C03658=1180.309,271.886,-67.108,-177.055,7.451,148.555
C03659=1180.314,271.637,-67.079,-177.057,7.448,148.555
C03660=1180.318,271.389,-67.051,-177.060,7.446,148.555
C03661=1180.323,271.140,-67.023,-177.063,7.443,148.555
C03662=1180.327,270.893,-66.995,-177.066,7.440,148.555
C03663=1180.331,270.644,-66.967,-177.068,7.438,148.555
C03664=1180.336,270.396,-66.938,-177.071,7.435,148.555
C03665=1180.340,270.147,-66.910,-177.073,7.432,148.555
C03666=1180.345,269.899,-66.882,-177.076,7.430,148.556
C03667=1180.348,269.651,-66.854,-177.078,7.427,148.556
C03668=1180.354,269.402,-66.825,-177.081,7.424,148.556
C03669=1180.357,269.154,-66.797,-177.083,7.421,148.556
C03670=1180.362,268.906,-66.769,-177.086,7.418,148.556
C03671=1180.366,268.657,-66.741,-177.089,7.416,148.556
C03672=1180.371,268.408,-66.714,-177.092,7.413,148.556
C03673=1180.375,268.160,-66.685,-177.094,7.411,148.556
C03674=1180.380,267.912,-66.657,-177.097,7.408,148.556
C03675=1180.383,267.663,-66.629,-177.099,7.405,148.556
C03676=1180.388,267.415,-66.601,-177.102,7.403,148.556
C03677=1180.393,267.167,-66.573,-177.104,7.400,148.556
C03678=1180.397,266.919,-66.545,-177.107,7.397,148.556
C03679=1180.401,266.670,-66.518,-177.109,7.394,148.557
C03680=1180.406,266.421,-66.489,-177.112,7.392,148.557
C03681=1180.410,266.173,-66.461,-177.115,7.389,148.557
C03682=1180.414,265.925,-66.433,-177.117,7.387,148.557
C03683=1180.419,265.676,-66.406,-177.120,7.384,148.557
C03684=1180.424,265.428,-66.378,-177.123,7.381,148.557
C03685=1180.427,265.179,-66.349,-177.125,7.379,148.557
C03686=1180.432,264.932,-66.322,-177.128,7.376,148.557
C03687=1180.436,264.682,-66.294,-177.131,7.373,148.557
C03688=1180.441,264.434,-66.266,-177.133,7.371,148.558
C03689=1180.445,264.186,-66.238,-177.136,7.368,148.558
C03690=1180.449,263.937,-66.211,-177.139,7.365,148.558
C03691=1180.454,263.689,-66.183,-177.141,7.363,148.558
C03692=1180.459,263.441,-66.154,-177.144,7.360,148.558
C03693=1180.463,263.192,-66.127,-177.146,7.357,148.558
C03694=1180.467,262.944,-66.099,-177.149,7.355,148.558
C03695=1180.472,262.671,-66.069,-177.152,7.352,148.558
C03696=1180.477,262.398,-66.038,-177.154,7.349,148.558
C03697=1180.481,262.125,-66.008,-177.157,7.346,148.558
C03698=1180.486,261.852,-65.978,-177.160,7.343,148.559
C03699=1180.490,261.604,-65.950,-177.163,7.340,148.559
C03700=1180.495,261.355,-65.922,-177.166,7.337,148.559
C03701=1180.500,261.107,-65.894,-177.168,7.335,148.559
C03702=1180.504,260.858,-65.867,-177.171,7.332,148.559
C03703=1180.508,260.610,-65.839,-177.173,7.330,148.559
C03704=1180.513,260.362,-65.812,-177.176,7.327,148.559
C03705=1180.517,260.113,-65.784,-177.179,7.324,148.559
C03706=1180.521,259.864,-65.757,-177.181,7.322,148.559
C03707=1180.526,259.617,-65.729,-177.184,7.319,148.559
C03708=1180.530,259.367,-65.702,-177.187,7.317,148.560
C03709=1180.534,259.119,-65.675,-177.189,7.314,148.560
C03710=1180.539,258.871,-65.647,-177.192,7.311,148.560
C03711=1180.543,258.623,-65.620,-177.194,7.309,148.560
C03712=1180.547,258.374,-65.592,-177.197,7.306,148.560
C03713=1180.552,258.125,-65.564,-177.200,7.304,148.560
C03714=1180.556,257.877,-65.537,-177.202,7.302,148.560
C03715=1180.561,257.629,-65.510,-177.205,7.299,148.560
C03716=1180.565,257.380,-65.482,-177.208,7.296,148.560
C03717=1180.569,257.131,-65.455,-177.210,7.293,148.560
C03718=1180.574,256.884,-65.427,-177.213,7.291,148.561
C03719=1180.578,256.635,-65.400,-177.215,7.289,148.561
C03720=1180.582,256.386,-65.373,-177.218,7.286,148.561
C03721=1180.587,256.138,-65.345,-177.221,7.283,148.561
C03722=1180.591,255.889,-65.318,-177.223,7.281,148.561
C03723=1180.596,255.641,-65.291,-177.226,7.278,148.561
C03724=1180.600,255.392,-65.264,-177.228,7.276,148.561
C03725=1180.604,255.144,-65.236,-177.231,7.273,148.561
C03726=1180.609,254.895,-65.209,-177.234,7.270,148.562
C03727=1180.614,254.647,-65.182,-177.236,7.268,148.562
C03728=1180.618,254.398,-65.155,-177.239,7.265,148.562
C03729=1180.623,254.150,-65.128,-177.241,7.263,148.562
C03730=1180.626,253.902,-65.100,-177.244,7.260,148.562
C03731=1180.631,253.653,-65.073,-177.247,7.257,148.562
C03732=1180.635,253.405,-65.046,-177.249,7.255,148.562
C03733=1180.640,253.156,-65.019,-177.252,7.252,148.562
C03734=1180.645,252.908,-64.992,-177.255,7.250,148.563
C03735=1180.649,252.658,-64.964,-177.257,7.247,148.563
C03736=1180.653,252.410,-64.937,-177.260,7.245,148.563
C03737=1180.657,252.162,-64.911,-177.262,7.242,148.563
C03738=1180.662,251.913,-64.884,-177.265,7.240,148.563
C03739=1180.667,251.665,-64.857,-177.268,7.237,148.563
C03740=1180.671,251.417,-64.829,-177.270,7.234,148.563
C03741=1180.676,251.168,-64.802,-177.273,7.233,148.564
C03742=1180.680,250.920,-64.775,-177.276,7.230,148.564
C03743=1180.684,250.671,-64.748,-177.278,7.227,148.564
C03744=1180.688,250.423,-64.721,-177.281,7.224,148.564
C03745=1180.693,250.174,-64.694,-177.284,7.222,148.564
C03746=1180.697,249.926,-64.667,-177.286,7.220,148.564
C03747=1180.702,249.677,-64.641,-177.289,7.217,148.564
C03748=1180.707,249.428,-64.614,-177.291,7.215,148.565
C03749=1180.711,249.180,-64.587,-177.294,7.212,148.565
C03750=1180.715,248.932,-64.560,-177.296,7.210,148.565
C03751=1180.720,248.683,-64.533,-177.299,7.207,148.565
C03752=1180.724,248.435,-64.506,-177.302,7.205,148.565
C03753=1180.728,248.186,-64.480,-177.304,7.202,148.565
C03754=1180.732,247.937,-64.452,-177.307,7.199,148.565
C03755=1180.737,247.689,-64.425,-177.310,7.197,148.566
C03756=1180.741,247.441,-64.399,-177.313,7.194,148.566
C03757=1180.746,247.191,-64.373,-177.315,7.192,148.566
C03758=1180.751,246.943,-64.345,-177.318,7.189,148.566
C03759=1180.755,246.695,-64.319,-177.320,7.187,148.566
C03760=1180.759,246.446,-64.292,-177.323,7.184,148.566
C03761=1180.764,246.198,-64.265,-177.326,7.182,148.567
C03762=1180.768,245.949,-64.239,-177.328,7.180,148.567
C03763=1180.773,245.700,-64.212,-177.330,7.177,148.567
C03764=1180.777,245.452,-64.185,-177.334,7.175,148.567
C03765=1180.781,245.204,-64.159,-177.336,7.173,148.567
C03766=1180.786,244.955,-64.132,-177.339,7.170,148.567
C03767=1180.790,244.706,-64.106,-177.342,7.167,148.567
C03768=1180.795,244.458,-64.079,-177.344,7.165,148.568
C03769=1180.799,244.209,-64.053,-177.347,7.162,148.568
C03770=1180.804,243.961,-64.026,-177.349,7.160,148.568
C03771=1180.808,243.712,-63.999,-177.352,7.157,148.568
C03772=1180.813,243.463,-63.973,-177.355,7.155,148.568
C03773=1180.817,243.215,-63.946,-177.357,7.152,148.568
C03774=1180.821,242.967,-63.920,-177.360,7.150,148.568
C03775=1180.826,242.718,-63.893,-177.363,7.147,148.569
C03776=1180.830,242.469,-63.867,-177.365,7.145,148.569
C03777=1180.835,242.220,-63.840,-177.368,7.142,148.569
C03778=1180.840,241.973,-63.814,-177.370,7.141,148.569
C03779=1180.844,241.724,-63.787,-177.373,7.138,148.569
C03780=1180.848,241.475,-63.761,-177.376,7.136,148.570
C03781=1180.852,241.227,-63.735,-177.379,7.133,148.570
C03782=1180.857,240.978,-63.709,-177.381,7.131,148.570
C03783=1180.861,240.730,-63.682,-177.384,7.128,148.570
C03784=1180.866,240.481,-63.656,-177.386,7.126,148.570
C03785=1180.870,240.233,-63.629,-177.389,7.123,148.570
C03786=1180.875,239.984,-63.603,-177.392,7.121,148.571
C03787=1180.879,239.735,-63.577,-177.394,7.118,148.571
C03788=1180.884,239.486,-63.550,-177.397,7.116,148.571
C03789=1180.889,239.238,-63.525,-177.400,7.113,148.571
C03790=1180.893,238.990,-63.498,-177.402,7.111,148.571
C03791=1180.898,238.741,-63.472,-177.405,7.109,148.571
C03792=1180.902,238.493,-63.446,-177.407,7.106,148.572
C03793=1180.906,238.244,-63.420,-177.410,7.104,148.572
C03794=1180.911,237.995,-63.393,-177.413,7.102,148.572
C03795=1180.915,237.747,-63.367,-177.415,7.100,148.572
C03796=1180.920,237.497,-63.341,-177.418,7.097,148.572
C03797=1180.924,237.249,-63.315,-177.421,7.095,148.573
C03798=1180.928,237.001,-63.289,-177.423,7.092,148.573
C03799=1180.933,236.729,-63.261,-177.427,7.089,148.573
C03800=1180.938,236.458,-63.231,-177.429,7.087,148.573
C03801=1180.943,236.186,-63.203,-177.432,7.085,148.573
C03802=1180.948,235.915,-63.175,-177.435,7.082,148.573
C03803=1180.953,235.666,-63.149,-177.437,7.080,148.574
C03804=1180.957,235.417,-63.123,-177.440,7.077,148.574
C03805=1180.961,235.168,-63.097,-177.443,7.075,148.574
C03806=1180.965,234.920,-63.071,-177.446,7.072,148.574
C03807=1180.970,234.671,-63.044,-177.448,7.070,148.575
C03808=1180.975,234.423,-63.019,-177.451,7.067,148.575
C03809=1180.979,234.174,-62.993,-177.454,7.065,148.575
C03810=1180.983,233.925,-62.967,-177.456,7.062,148.575
C03811=1180.988,233.677,-62.940,-177.458,7.060,148.575
C03812=1180.993,233.429,-62.915,-177.462,7.058,148.575
C03813=1180.997,233.180,-62.889,-177.464,7.056,148.576
C03814=1181.001,232.931,-62.863,-177.467,7.054,148.576
C03815=1181.006,232.682,-62.838,-177.469,7.051,148.576
C03816=1181.011,232.434,-62.812,-177.472,7.049,148.576
C03817=1181.015,232.185,-62.786,-177.475,7.046,148.576
C03818=1181.020,231.936,-62.760,-177.477,7.044,148.577
C03819=1181.024,231.688,-62.734,-177.480,7.041,148.577
C03820=1181.028,231.440,-62.708,-177.483,7.039,148.577
C03821=1181.033,231.191,-62.683,-177.485,7.037,148.577
C03822=1181.038,230.942,-62.656,-177.488,7.035,148.577
C03823=1181.042,230.693,-62.631,-177.490,7.032,148.578
C03824=1181.047,230.445,-62.605,-177.493,7.030,148.578
C03825=1181.051,230.196,-62.579,-177.496,7.028,148.578
C03826=1181.055,229.948,-62.554,-177.499,7.025,148.578
C03827=1181.060,229.700,-62.528,-177.501,7.023,148.578
C03828=1181.064,229.451,-62.503,-177.504,7.021,148.579
C03829=1181.068,229.202,-62.477,-177.506,7.018,148.579
C03830=1181.073,228.953,-62.452,-177.509,7.016,148.579
C03831=1181.078,228.704,-62.426,-177.512,7.013,148.579
C03832=1181.082,228.456,-62.401,-177.515,7.012,148.580
C03833=1181.087,228.208,-62.375,-177.517,7.009,148.580
C03834=1181.092,227.958,-62.349,-177.520,7.007,148.580
C03835=1181.096,227.710,-62.323,-177.522,7.005,148.580
C03836=1181.101,227.462,-62.298,-177.525,7.002,148.580
C03837=1181.105,227.213,-62.272,-177.528,7.000,148.581
C03838=1181.109,226.964,-62.246,-177.530,6.998,148.581
C03839=1181.114,226.715,-62.222,-177.533,6.995,148.581
C03840=1181.119,226.466,-62.196,-177.536,6.993,148.581
C03841=1181.123,226.218,-62.170,-177.539,6.991,148.581
C03842=1181.128,225.969,-62.145,-177.541,6.989,148.582
C03843=1181.131,225.721,-62.120,-177.544,6.987,148.582
C03844=1181.136,225.472,-62.095,-177.546,6.984,148.582
C03845=1181.140,225.223,-62.069,-177.549,6.982,148.582
C03846=1181.145,224.975,-62.043,-177.552,6.979,148.582
C03847=1181.149,224.727,-62.018,-177.554,6.977,148.583
C03848=1181.154,224.477,-61.993,-177.557,6.975,148.583
C03849=1181.159,224.229,-61.968,-177.560,6.972,148.583
C03850=1181.163,223.980,-61.942,-177.562,6.971,148.583
C03851=1181.168,223.731,-61.917,-177.565,6.968,148.584
C03852=1181.172,223.483,-61.891,-177.568,6.966,148.584
C03853=1181.177,223.234,-61.866,-177.570,6.964,148.584
C03854=1181.182,222.985,-61.841,-177.573,6.961,148.584
C03855=1181.185,222.737,-61.816,-177.576,6.959,148.585
C03856=1181.190,222.489,-61.790,-177.578,6.957,148.585
C03857=1181.195,222.239,-61.765,-177.581,6.954,148.585
C03858=1181.199,221.990,-61.740,-177.583,6.952,148.585
C03859=1181.204,221.742,-61.715,-177.586,6.951,148.585
C03860=1181.208,221.493,-61.689,-177.589,6.948,148.586
C03861=1181.213,221.244,-61.665,-177.592,6.946,148.586
C03862=1181.217,220.996,-61.639,-177.594,6.944,148.586
C03863=1181.222,220.747,-61.614,-177.597,6.941,148.586
C03864=1181.226,220.498,-61.589,-177.600,6.939,148.587
C03865=1181.231,220.250,-61.564,-177.602,6.936,148.587
C03866=1181.235,220.001,-61.539,-177.605,6.934,148.587
C03867=1181.240,219.753,-61.514,-177.608,6.933,148.587
C03868=1181.244,219.503,-61.489,-177.610,6.930,148.587
C03869=1181.249,219.255,-61.463,-177.613,6.928,148.588
C03870=1181.254,219.006,-61.438,-177.616,6.926,148.588
C03871=1181.258,218.757,-61.414,-177.618,6.923,148.588
C03872=1181.262,218.509,-61.388,-177.621,6.921,148.589
C03873=1181.267,218.260,-61.364,-177.623,6.919,148.589
C03874=1181.271,218.011,-61.339,-177.627,6.917,148.589
C03875=1181.276,217.763,-61.314,-177.629,6.915,148.589
C03876=1181.280,217.514,-61.288,-177.631,6.913,148.589
C03877=1181.285,217.265,-61.264,-177.635,6.910,148.590
C03878=1181.290,217.017,-61.239,-177.637,6.908,148.590
C03879=1181.294,216.768,-61.214,-177.639,6.906,148.590
C03880=1181.299,216.519,-61.189,-177.643,6.903,148.590
C03881=1181.303,216.270,-61.165,-177.645,6.901,148.591
C03882=1181.308,216.022,-61.139,-177.648,6.899,148.591
C03883=1181.312,215.773,-61.114,-177.651,6.897,148.591
C03884=1181.317,215.524,-61.090,-177.653,6.895,148.591
C03885=1181.322,215.275,-61.065,-177.656,6.893,148.592
C03886=1181.325,215.027,-61.040,-177.659,6.890,148.592
C03887=1181.330,214.778,-61.016,-177.661,6.888,148.592
C03888=1181.335,214.529,-60.991,-177.664,6.886,148.592
C03889=1181.339,214.280,-60.967,-177.667,6.884,148.593
C03890=1181.344,214.032,-60.941,-177.669,6.882,148.593
C03891=1181.348,213.783,-60.917,-177.672,6.880,148.593
C03892=1181.353,213.534,-60.892,-177.674,6.878,148.594
C03893=1181.357,213.285,-60.867,-177.677,6.875,148.594
C03894=1181.362,213.037,-60.843,-177.680,6.873,148.594
C03895=1181.367,212.788,-60.818,-177.682,6.871,148.594
C03896=1181.371,212.539,-60.793,-177.685,6.868,148.594
C03897=1181.376,212.291,-60.768,-177.688,6.867,148.595
C03898=1181.380,212.042,-60.744,-177.691,6.865,148.595
C03899=1181.385,211.793,-60.719,-177.693,6.862,148.595
C03900=1181.389,211.544,-60.695,-177.696,6.860,148.596
C03901=1181.394,211.296,-60.671,-177.699,6.858,148.596
C03902=1181.398,211.047,-60.646,-177.701,6.856,148.596
C03903=1181.403,210.776,-60.619,-177.704,6.854,148.596
C03904=1181.408,210.506,-60.593,-177.707,6.851,148.597
C03905=1181.413,210.235,-60.566,-177.710,6.849,148.597
C03906=1181.418,209.965,-60.539,-177.713,6.846,148.597
C03907=1181.422,209.717,-60.515,-177.715,6.844,148.597
C03908=1181.427,209.467,-60.490,-177.718,6.843,148.598
C03909=1181.431,209.219,-60.466,-177.721,6.840,148.598
C03910=1181.436,208.970,-60.441,-177.723,6.838,148.598
C03911=1181.441,208.722,-60.417,-177.726,6.836,148.598
C03912=1181.445,208.472,-60.392,-177.729,6.834,148.599
C03913=1181.450,208.224,-60.368,-177.731,6.831,148.599
C03914=1181.454,207.975,-60.345,-177.734,6.829,148.599
C03915=1181.459,207.726,-60.320,-177.737,6.828,148.600
C03916=1181.463,207.477,-60.295,-177.739,6.826,148.600
C03917=1181.468,207.228,-60.271,-177.742,6.823,148.600
C03918=1181.473,206.980,-60.247,-177.745,6.821,148.600
C03919=1181.477,206.732,-60.223,-177.748,6.819,148.601
C03920=1181.482,206.482,-60.198,-177.750,6.816,148.601
C03921=1181.486,206.234,-60.173,-177.753,6.815,148.601
C03922=1181.491,205.985,-60.150,-177.756,6.813,148.601
C03923=1181.496,205.736,-60.125,-177.758,6.811,148.602
C03924=1181.500,205.487,-60.101,-177.761,6.808,148.602
C03925=1181.504,205.238,-60.077,-177.764,6.806,148.602
C03926=1181.509,204.990,-60.052,-177.766,6.804,148.603
C03927=1181.514,204.741,-60.029,-177.769,6.802,148.603
C03928=1181.518,204.492,-60.005,-177.772,6.800,148.603
C03929=1181.523,204.243,-59.980,-177.774,6.798,148.603
C03930=1181.527,203.994,-59.956,-177.777,6.796,148.604
C03931=1181.532,203.745,-59.932,-177.779,6.794,148.604
C03932=1181.536,203.497,-59.908,-177.782,6.791,148.604
C03933=1181.542,203.248,-59.884,-177.785,6.789,148.605
C03934=1181.545,202.999,-59.859,-177.788,6.788,148.605
C03935=1181.550,202.750,-59.836,-177.790,6.786,148.605
C03936=1181.554,202.502,-59.812,-177.793,6.784,148.605
C03937=1181.560,202.253,-59.787,-177.796,6.781,148.606
C03938=1181.564,202.004,-59.764,-177.798,6.779,148.606
C03939=1181.569,201.755,-59.740,-177.801,6.777,148.606
C03940=1181.573,201.507,-59.716,-177.803,6.775,148.606
C03941=1181.577,201.257,-59.692,-177.807,6.773,148.607
C03942=1181.582,201.009,-59.667,-177.809,6.771,148.607
C03943=1181.587,200.760,-59.644,-177.812,6.769,148.607
C03944=1181.591,200.511,-59.620,-177.814,6.767,148.608
C03945=1181.596,200.263,-59.596,-177.817,6.765,148.608
C03946=1181.600,200.014,-59.572,-177.820,6.763,148.608
C03947=1181.605,199.765,-59.548,-177.822,6.761,148.608
C03948=1181.610,199.516,-59.525,-177.825,6.759,148.609
C03949=1181.614,199.267,-59.500,-177.828,6.757,148.609
C03950=1181.619,199.018,-59.476,-177.831,6.754,148.609
C03951=1181.623,198.769,-59.452,-177.833,6.752,148.610
C03952=1181.628,198.520,-59.429,-177.836,6.750,148.610
C03953=1181.632,198.272,-59.405,-177.838,6.749,148.610
C03954=1181.637,198.023,-59.382,-177.841,6.747,148.611
C03955=1181.641,197.775,-59.358,-177.844,6.744,148.611
C03956=1181.646,197.525,-59.334,-177.846,6.742,148.611
C03957=1181.651,197.276,-59.311,-177.849,6.740,148.611
C03958=1181.655,197.028,-59.287,-177.852,6.739,148.612
C03959=1181.660,196.779,-59.263,-177.854,6.737,148.612
C03960=1181.665,196.530,-59.239,-177.857,6.735,148.612
C03961=1181.670,196.281,-59.215,-177.860,6.732,148.613
C03962=1181.674,196.032,-59.192,-177.863,6.730,148.613
C03963=1181.679,195.784,-59.168,-177.865,6.728,148.613
C03964=1181.683,195.535,-59.145,-177.868,6.727,148.614
C03965=1181.688,195.286,-59.121,-177.870,6.724,148.614
C03966=1181.692,195.037,-59.097,-177.873,6.722,148.614
C03967=1181.697,194.788,-59.073,-177.876,6.720,148.614
C03968=1181.701,194.539,-59.050,-177.879,6.718,148.615
C03969=1181.706,194.290,-59.026,-177.881,6.716,148.615
C03970=1181.710,194.041,-59.003,-177.883,6.714,148.615
C03971=1181.715,193.792,-58.979,-177.886,6.713,148.616
C03972=1181.719,193.545,-58.956,-177.889,6.710,148.616
C03973=1181.724,193.296,-58.933,-177.892,6.708,148.616
C03974=1181.729,193.047,-58.909,-177.895,6.706,148.617
C03975=1181.734,192.798,-58.886,-177.897,6.704,148.617
C03976=1181.738,192.549,-58.863,-177.900,6.702,148.617
C03977=1181.743,192.300,-58.839,-177.902,6.701,148.617
C03978=1181.747,192.051,-58.815,-177.905,6.698,148.618
C03979=1181.752,191.802,-58.792,-177.908,6.696,148.618
C03980=1181.757,191.553,-58.769,-177.911,6.694,148.618
C03981=1181.761,191.304,-58.745,-177.913,6.692,148.619
C03982=1181.766,191.055,-58.722,-177.916,6.691,148.619
C03983=1181.771,190.807,-58.698,-177.918,6.689,148.619
C03984=1181.774,190.558,-58.675,-177.922,6.686,148.620
C03985=1181.779,190.309,-58.652,-177.924,6.684,148.620
C03986=1181.784,190.060,-58.628,-177.927,6.683,148.620
C03987=1181.789,189.811,-58.605,-177.929,6.680,148.620
C03988=1181.793,189.562,-58.582,-177.932,6.679,148.621
C03989=1181.798,189.313,-58.558,-177.934,6.677,148.621
C03990=1181.803,189.065,-58.536,-177.937,6.675,148.622
C03991=1181.807,188.816,-58.512,-177.940,6.672,148.622
C03992=1181.812,188.567,-58.489,-177.943,6.671,148.622
C03993=1181.817,188.318,-58.466,-177.945,6.669,148.622
C03994=1181.821,188.069,-58.442,-177.948,6.667,148.623
C03995=1181.825,187.820,-58.420,-177.951,6.665,148.623
C03996=1181.830,187.571,-58.396,-177.953,6.663,148.623
C03997=1181.835,187.322,-58.373,-177.956,6.661,148.624
C03998=1181.840,187.073,-58.350,-177.959,6.660,148.624
C03999=1181.844,186.825,-58.327,-177.962,6.657,148.624
C04000=1181.849,186.576,-58.304,-177.964,6.655,148.625
C04001=1181.853,186.327,-58.280,-177.967,6.653,148.625
C04002=1181.858,186.078,-58.257,-177.969,6.651,148.625
C04003=1181.862,185.829,-58.234,-177.972,6.650,148.626
C04004=1181.867,185.580,-58.211,-177.975,6.648,148.626
C04005=1181.872,185.332,-58.188,-177.977,6.646,148.626
C04006=1181.876,185.082,-58.166,-177.980,6.644,148.627
C04007=1181.881,184.813,-58.140,-177.983,6.642,148.627
C04008=1181.887,184.543,-58.115,-177.986,6.640,148.627
C04009=1181.891,184.274,-58.091,-177.989,6.638,148.628
C04010=1181.897,184.004,-58.066,-177.992,6.635,148.628
C04011=1181.901,183.755,-58.042,-177.995,6.634,148.628
C04012=1181.905,183.506,-58.020,-177.997,6.632,148.629
C04013=1181.910,183.257,-57.997,-177.999,6.630,148.629
C04014=1181.915,183.008,-57.974,-178.002,6.628,148.629
C04015=1181.919,182.760,-57.951,-178.005,6.626,148.630
C04016=1181.924,182.511,-57.928,-178.007,6.624,148.630
C04017=1181.928,182.261,-57.906,-178.010,6.623,148.630
C04018=1181.933,182.012,-57.882,-178.013,6.620,148.631
C04019=1181.938,181.764,-57.859,-178.016,6.618,148.631
C04020=1181.943,181.515,-57.837,-178.019,6.616,148.631
C04021=1181.947,181.265,-57.814,-178.021,6.615,148.632
C04022=1181.951,181.017,-57.791,-178.024,6.613,148.632
C04023=1181.957,180.768,-57.768,-178.026,6.611,148.632
C04024=1181.961,180.519,-57.746,-178.029,6.609,148.633
C04025=1181.966,180.270,-57.723,-178.032,6.607,148.633
C04026=1181.970,180.021,-57.701,-178.034,6.605,148.633
C04027=1181.975,179.772,-57.678,-178.037,6.604,148.634
C04028=1181.979,179.524,-57.655,-178.040,6.602,148.634
C04029=1181.984,179.274,-57.632,-178.042,6.600,148.634
C04030=1181.989,179.026,-57.609,-178.046,6.597,148.635
C04031=1181.993,178.777,-57.587,-178.048,6.596,148.635
C04032=1181.998,178.527,-57.564,-178.051,6.594,148.635
C04033=1182.002,178.279,-57.541,-178.053,6.592,148.636
C04034=1182.007,178.030,-57.519,-178.056,6.590,148.636
C04035=1182.012,177.781,-57.496,-178.058,6.588,148.636
C04036=1182.016,177.532,-57.474,-178.061,6.586,148.637
C04037=1182.022,177.283,-57.451,-178.064,6.585,148.637
C04038=1182.026,177.034,-57.429,-178.066,6.583,148.637
C04039=1182.030,176.785,-57.406,-178.069,6.581,148.638
C04040=1182.035,176.536,-57.384,-178.072,6.579,148.638
C04041=1182.040,176.287,-57.361,-178.074,6.578,148.638
C04042=1182.044,176.038,-57.339,-178.077,6.576,148.639
C04043=1182.049,175.790,-57.316,-178.080,6.574,148.639
C04044=1182.054,175.540,-57.294,-178.083,6.572,148.640
C04045=1182.058,175.291,-57.271,-178.085,6.570,148.640
C04046=1182.063,175.043,-57.248,-178.088,6.569,148.640
C04047=1182.068,174.793,-57.226,-178.091,6.567,148.641
C04048=1182.072,174.545,-57.204,-178.093,6.565,148.641
C04049=1182.077,174.295,-57.181,-178.095,6.563,148.641
C04050=1182.082,174.046,-57.159,-178.099,6.560,148.642
C04051=1182.086,173.798,-57.137,-178.101,6.559,148.642
C04052=1182.091,173.548,-57.114,-178.104,6.557,148.642
C04053=1182.096,173.300,-57.092,-178.107,6.555,148.643
C04054=1182.100,173.051,-57.070,-178.109,6.553,148.643
C04055=1182.105,172.801,-57.047,-178.112,6.551,148.643
C04056=1182.110,172.553,-57.026,-178.115,6.550,148.644
C04057=1182.114,172.304,-57.003,-178.117,6.548,148.644
C04058=1182.119,172.055,-56.981,-178.120,6.546,148.644
C04059=1182.124,171.806,-56.958,-178.123,6.544,148.645
C04060=1182.128,171.558,-56.936,-178.125,6.543,148.645
C04061=1182.133,171.308,-56.913,-178.128,6.541,148.646
C04062=1182.138,171.059,-56.891,-178.131,6.539,148.646
C04063=1182.142,170.810,-56.870,-178.133,6.537,148.646
C04064=1182.146,170.561,-56.847,-178.136,6.535,148.647
C04065=1182.152,170.312,-56.825,-178.139,6.534,148.647
C04066=1182.156,170.063,-56.803,-178.141,6.532,148.647
C04067=1182.161,169.815,-56.781,-178.144,6.530,148.648
C04068=1182.165,169.565,-56.759,-178.147,6.528,148.648
C04069=1182.171,169.316,-56.737,-178.150,6.527,148.648
C04070=1182.175,169.067,-56.714,-178.152,6.525,148.649
C04071=1182.180,168.819,-56.692,-178.155,6.523,148.649
C04072=1182.184,168.570,-56.670,-178.158,6.521,148.650
C04073=1182.189,168.321,-56.648,-178.160,6.520,148.650
C04074=1182.194,168.071,-56.626,-178.163,6.518,148.650
C04075=1182.199,167.823,-56.604,-178.166,6.516,148.651
C04076=1182.203,167.573,-56.582,-178.168,6.514,148.651
C04077=1182.208,167.325,-56.560,-178.171,6.512,148.651
C04078=1182.212,167.075,-56.538,-178.174,6.511,148.652
C04079=1182.217,166.827,-56.517,-178.176,6.509,148.652
C04080=1182.222,166.577,-56.494,-178.179,6.507,148.652
C04081=1182.227,166.328,-56.472,-178.182,6.505,148.653
C04082=1182.231,166.080,-56.450,-178.184,6.504,148.653
C04083=1182.236,165.831,-56.428,-178.187,6.502,148.654
C04084=1182.240,165.582,-56.406,-178.190,6.500,148.654
C04085=1182.245,165.332,-56.385,-178.192,6.498,148.654
C04086=1182.250,165.083,-56.363,-178.195,6.496,148.655
C04087=1182.254,164.834,-56.341,-178.198,6.495,148.655
C04088=1182.259,164.586,-56.319,-178.200,6.493,148.655
C04089=1182.264,164.336,-56.297,-178.203,6.492,148.656
C04090=1182.268,164.088,-56.276,-178.205,6.490,148.656
C04091=1182.273,163.838,-56.254,-178.208,6.488,148.657
C04092=1182.278,163.589,-56.231,-178.211,6.487,148.657
C04093=1182.283,163.340,-56.209,-178.213,6.485,148.657
C04094=1182.287,163.091,-56.188,-178.216,6.483,148.658
C04095=1182.292,162.843,-56.166,-178.219,6.481,148.658
C04096=1182.297,162.593,-56.144,-178.221,6.480,148.658
C04097=1182.302,162.344,-56.123,-178.224,6.478,148.659
C04098=1182.306,162.095,-56.101,-178.227,6.476,148.659
C04099=1182.311,161.846,-56.079,-178.229,6.474,148.660
C04100=1182.316,161.598,-56.058,-178.232,6.472,148.660
C04101=1182.320,161.348,-56.035,-178.235,6.471,148.660
C04102=1182.325,161.100,-56.014,-178.237,6.469,148.661
C04103=1182.330,160.850,-55.993,-178.240,6.467,148.661
C04104=1182.334,160.601,-55.971,-178.243,6.465,148.661
C04105=1182.338,160.353,-55.950,-178.245,6.464,148.662
C04106=1182.343,160.103,-55.928,-178.248,6.462,148.662
C04107=1182.348,159.854,-55.907,-178.251,6.460,148.663
C04108=1182.353,159.605,-55.885,-178.254,6.459,148.663
C04109=1182.357,159.356,-55.863,-178.256,6.458,148.664
C04110=1182.362,159.107,-55.841,-178.259,6.456,148.664
C04111=1182.367,158.838,-55.818,-178.262,6.453,148.664
C04112=1182.372,158.569,-55.795,-178.265,6.452,148.665
C04113=1182.378,158.300,-55.772,-178.267,6.450,148.665
C04114=1182.382,158.031,-55.748,-178.271,6.448,148.666
C04115=1182.387,157.782,-55.727,-178.273,6.447,148.666
C04116=1182.392,157.533,-55.706,-178.276,6.445,148.666
C04117=1182.396,157.284,-55.684,-178.279,6.443,148.667
C04118=1182.402,157.035,-55.663,-178.281,6.441,148.667
C04119=1182.406,156.786,-55.642,-178.284,6.440,148.667
C04120=1182.411,156.537,-55.621,-178.287,6.438,148.668
C04121=1182.415,156.288,-55.599,-178.289,6.437,148.668
C04122=1182.420,156.039,-55.577,-178.292,6.435,148.669
C04123=1182.425,155.790,-55.556,-178.294,6.433,148.669
C04124=1182.429,155.541,-55.534,-178.297,6.432,148.669
C04125=1182.434,155.292,-55.513,-178.300,6.430,148.670
C04126=1182.439,155.043,-55.492,-178.302,6.428,148.670
C04127=1182.444,154.794,-55.471,-178.305,6.427,148.671
C04128=1182.448,154.544,-55.449,-178.308,6.425,148.671
C04129=1182.453,154.295,-55.428,-178.311,6.423,148.671
C04130=1182.457,154.047,-55.407,-178.313,6.421,148.672
C04131=1182.463,153.798,-55.386,-178.316,6.420,148.672
C04132=1182.467,153.549,-55.364,-178.318,6.419,148.673
C04133=1182.471,153.299,-55.343,-178.321,6.417,148.673
C04134=1182.476,153.051,-55.322,-178.324,6.415,148.673
C04135=1182.481,152.801,-55.301,-178.326,6.413,148.674
C04136=1182.486,152.553,-55.279,-178.329,6.412,148.674
C04137=1182.490,152.303,-55.258,-178.332,6.410,148.675
C04138=1182.495,152.054,-55.237,-178.335,6.408,148.675
C04139=1182.500,151.805,-55.216,-178.338,6.407,148.675
C04140=1182.505,151.556,-55.195,-178.340,6.406,148.676
C04141=1182.509,151.308,-55.174,-178.342,6.404,148.676
C04142=1182.515,151.058,-55.153,-178.345,6.402,148.677
C04143=1182.519,150.808,-55.131,-178.348,6.400,148.677
C04144=1182.523,150.560,-55.110,-178.350,6.399,148.677
C04145=1182.528,150.311,-55.089,-178.353,6.397,148.678
C04146=1182.534,150.062,-55.068,-178.356,6.395,148.678
C04147=1182.538,149.813,-55.047,-178.358,6.394,148.679
C04148=1182.543,149.564,-55.026,-178.361,6.393,148.679
C04149=1182.547,149.314,-55.005,-178.364,6.391,148.680
C04150=1182.552,149.065,-54.984,-178.366,6.389,148.680
C04151=1182.557,148.816,-54.963,-178.369,6.387,148.680
C04152=1182.561,148.567,-54.942,-178.372,6.386,148.681
C04153=1182.566,148.318,-54.921,-178.375,6.384,148.681
C04154=1182.571,148.069,-54.901,-178.377,6.382,148.681
C04155=1182.576,147.821,-54.879,-178.380,6.382,148.682
C04156=1182.580,147.571,-54.858,-178.383,6.380,148.682
C04157=1182.585,147.322,-54.838,-178.385,6.378,148.683
C04158=1182.590,147.072,-54.817,-178.388,6.376,148.683
C04159=1182.594,146.823,-54.796,-178.391,6.375,148.684
C04160=1182.599,146.575,-54.775,-178.393,6.373,148.684
C04161=1182.604,146.326,-54.754,-178.395,6.372,148.684
C04162=1182.609,146.077,-54.733,-178.399,6.370,148.685
C04163=1182.613,145.828,-54.713,-178.401,6.369,148.685
C04164=1182.618,145.578,-54.692,-178.404,6.367,148.686
C04165=1182.623,145.329,-54.672,-178.407,6.365,148.686
C04166=1182.628,145.080,-54.651,-178.409,6.363,148.686
C04167=1182.632,144.831,-54.630,-178.411,6.362,148.687
C04168=1182.637,144.582,-54.608,-178.414,6.361,148.687
C04169=1182.641,144.333,-54.588,-178.417,6.359,148.688
C04170=1182.646,144.084,-54.567,-178.420,6.357,148.688
C04171=1182.651,143.835,-54.547,-178.423,6.356,148.689
C04172=1182.656,143.586,-54.526,-178.425,6.354,148.689
C04173=1182.660,143.337,-54.505,-178.427,6.353,148.689
C04174=1182.666,143.087,-54.484,-178.430,6.351,148.690
C04175=1182.670,142.838,-54.464,-178.433,6.350,148.690
C04176=1182.675,142.589,-54.443,-178.436,6.348,148.691
C04177=1182.680,142.340,-54.423,-178.439,6.346,148.691
C04178=1182.684,142.091,-54.402,-178.441,6.345,148.692
C04179=1182.689,141.842,-54.381,-178.444,6.344,148.692
C04180=1182.694,141.593,-54.361,-178.446,6.342,148.692
C04181=1182.699,141.344,-54.340,-178.449,6.340,148.693
C04182=1182.703,141.095,-54.319,-178.452,6.339,148.693
C04183=1182.708,140.846,-54.299,-178.455,6.337,148.694
C04184=1182.713,140.596,-54.279,-178.457,6.336,148.694
C04185=1182.718,140.347,-54.258,-178.460,6.334,148.694
C04186=1182.722,140.098,-54.238,-178.462,6.333,148.695
C04187=1182.727,139.849,-54.217,-178.465,6.331,148.695
C04188=1182.732,139.600,-54.197,-178.468,6.329,148.696
C04189=1182.736,139.351,-54.176,-178.470,6.328,148.696
C04190=1182.741,139.102,-54.155,-178.473,6.327,148.697
C04191=1182.746,138.853,-54.135,-178.476,6.325,148.697
C04192=1182.751,138.603,-54.115,-178.479,6.324,148.698
C04193=1182.756,138.354,-54.094,-178.482,6.322,148.698
C04194=1182.760,138.105,-54.074,-178.484,6.321,148.698
C04195=1182.765,137.856,-54.054,-178.486,6.319,148.699
C04196=1182.770,137.607,-54.033,-178.489,6.317,148.699
C04197=1182.775,137.357,-54.013,-178.492,6.316,148.700
C04198=1182.780,137.109,-53.993,-178.494,6.315,148.700
C04199=1182.784,136.860,-53.973,-178.497,6.313,148.701
C04200=1182.789,136.611,-53.952,-178.500,6.311,148.701
C04201=1182.794,136.361,-53.932,-178.502,6.310,148.701
C04202=1182.798,136.112,-53.912,-178.506,6.308,148.702
C04203=1182.803,135.863,-53.891,-178.508,6.307,148.702
C04204=1182.808,135.614,-53.870,-178.510,6.306,148.703
C04205=1182.813,135.364,-53.851,-178.513,6.304,148.703
C04206=1182.817,135.115,-53.830,-178.516,6.302,148.704
C04207=1182.822,134.866,-53.810,-178.518,6.302,148.704
C04208=1182.828,134.617,-53.790,-178.521,6.300,148.705
C04209=1182.832,134.368,-53.770,-178.524,6.298,148.705
C04210=1182.837,134.119,-53.749,-178.527,6.296,148.705
C04211=1182.841,133.870,-53.730,-178.529,6.295,148.706
C04212=1182.846,133.621,-53.709,-178.532,6.294,148.706
C04213=1182.850,133.371,-53.690,-178.535,6.292,148.707
C04214=1182.856,133.122,-53.669,-178.537,6.290,148.707
C04215=1182.861,132.853,-53.648,-178.540,6.289,148.708
C04216=1182.866,132.585,-53.625,-178.543,6.287,148.708
C04217=1182.871,132.316,-53.604,-178.546,6.286,148.709
C04218=1182.876,132.048,-53.582,-178.549,6.284,148.709
C04219=1182.881,131.799,-53.562,-178.551,6.283,148.710
C04220=1182.886,131.550,-53.542,-178.554,6.281,148.710
C04221=1182.891,131.301,-53.522,-178.556,6.280,148.710
C04222=1182.895,131.052,-53.502,-178.560,6.278,148.711
C04223=1182.900,130.802,-53.482,-178.562,6.277,148.711
C04224=1182.904,130.553,-53.462,-178.564,6.276,148.712
C04225=1182.910,130.304,-53.443,-178.567,6.274,148.712
C04226=1182.914,130.055,-53.422,-178.570,6.273,148.713
C04227=1182.919,129.806,-53.403,-178.572,6.272,148.713
C04228=1182.924,129.556,-53.382,-178.575,6.270,148.714
C04229=1182.929,129.307,-53.362,-178.578,6.268,148.714
C04230=1182.934,129.058,-53.343,-178.580,6.267,148.715
C04231=1182.939,128.809,-53.322,-178.583,6.266,148.715
C04232=1182.943,128.560,-53.303,-178.586,6.264,148.715
C04233=1182.948,128.311,-53.282,-178.589,6.262,148.716
C04234=1182.953,128.062,-53.263,-178.591,6.262,148.716
C04235=1182.958,127.812,-53.243,-178.594,6.260,148.717
C04236=1182.962,127.563,-53.223,-178.597,6.258,148.717
C04237=1182.967,127.314,-53.203,-178.599,6.257,148.718
C04238=1182.972,127.065,-53.184,-178.602,6.256,148.718
C04239=1182.977,126.816,-53.164,-178.605,6.254,148.719
C04240=1182.981,126.566,-53.144,-178.607,6.252,148.719
C04241=1182.986,126.317,-53.124,-178.609,6.251,148.719
C04242=1182.991,126.069,-53.104,-178.613,6.250,148.720
C04243=1182.996,125.819,-53.085,-178.615,6.248,148.720
C04244=1183.000,125.570,-53.066,-178.617,6.247,148.721
C04245=1183.004,125.321,-53.045,-178.620,6.246,148.721
C04246=1183.010,125.072,-53.026,-178.623,6.244,148.722
C04247=1183.015,124.822,-53.006,-178.625,6.243,148.722
C04248=1183.019,124.573,-52.987,-178.628,6.242,148.723
C04249=1183.024,124.325,-52.967,-178.631,6.240,148.723
C04250=1183.029,124.075,-52.947,-178.634,6.238,148.724
C04251=1183.034,123.825,-52.927,-178.636,6.237,148.724
C04252=1183.039,123.577,-52.908,-178.639,6.236,148.724
C04253=1183.044,123.327,-52.888,-178.642,6.234,148.725
C04254=1183.048,123.078,-52.868,-178.644,6.233,148.726
C04255=1183.053,122.829,-52.849,-178.647,6.232,148.726
C04256=1183.058,122.580,-52.830,-178.650,6.230,148.727
C04257=1183.062,122.330,-52.810,-178.652,6.229,148.727
C04258=1183.068,122.081,-52.791,-178.655,6.228,148.727
C04259=1183.073,121.832,-52.771,-178.658,6.226,148.728
C04260=1183.077,121.583,-52.751,-178.660,6.225,148.728
C04261=1183.082,121.334,-52.732,-178.663,6.224,148.729
C04262=1183.086,121.085,-52.712,-178.666,6.222,148.729
C04263=1183.091,120.835,-52.693,-178.668,6.221,148.730
C04264=1183.096,120.586,-52.673,-178.671,6.219,148.730
C04265=1183.101,120.337,-52.654,-178.674,6.218,148.731
C04266=1183.105,120.088,-52.635,-178.676,6.217,148.731
C04267=1183.110,119.839,-52.615,-178.679,6.215,148.732
C04268=1183.115,119.589,-52.596,-178.682,6.214,148.732
C04269=1183.121,119.340,-52.576,-178.684,6.213,148.732
C04270=1183.125,119.091,-52.557,-178.687,6.211,148.733
C04271=1183.129,118.841,-52.538,-178.690,6.210,148.733
C04272=1183.135,118.593,-52.518,-178.692,6.209,148.734
C04273=1183.139,118.343,-52.499,-178.695,6.207,148.734
C04274=1183.145,118.094,-52.480,-178.698,6.206,148.735
C04275=1183.149,117.845,-52.460,-178.700,6.205,148.735
C04276=1183.154,117.596,-52.441,-178.703,6.203,148.736
C04277=1183.159,117.346,-52.422,-178.706,6.201,148.736
C04278=1183.163,117.097,-52.402,-178.708,6.201,148.737
C04279=1183.168,116.848,-52.383,-178.711,6.199,148.737
C04280=1183.173,116.599,-52.364,-178.714,6.197,148.738
C04281=1183.178,116.350,-52.344,-178.716,6.197,148.738
C04282=1183.182,116.101,-52.325,-178.718,6.195,148.739
C04283=1183.188,115.852,-52.306,-178.721,6.194,148.739
C04284=1183.193,115.602,-52.287,-178.724,6.192,148.740
C04285=1183.197,115.353,-52.268,-178.727,6.191,148.740
C04286=1183.202,115.103,-52.249,-178.729,6.190,148.741
C04287=1183.207,114.855,-52.229,-178.732,6.188,148.741
C04288=1183.211,114.605,-52.210,-178.735,6.187,148.741
C04289=1183.217,114.356,-52.191,-178.737,6.186,148.742
C04290=1183.221,114.107,-52.173,-178.740,6.184,148.742
C04291=1183.226,113.858,-52.153,-178.742,6.183,148.743
C04292=1183.231,113.608,-52.134,-178.745,6.182,148.744
C04293=1183.236,113.360,-52.115,-178.748,6.180,148.744
C04294=1183.240,113.110,-52.095,-178.750,6.179,148.744
C04295=1183.245,112.861,-52.077,-178.753,6.178,148.745
C04296=1183.250,112.611,-52.058,-178.756,6.176,148.745
C04297=1183.255,112.362,-52.038,-178.758,6.175,148.746
C04298=1183.259,112.113,-52.019,-178.761,6.174,148.746
C04299=1183.265,111.864,-52.001,-178.763,6.173,148.747
C04300=1183.269,111.614,-51.982,-178.767,6.172,148.747
C04301=1183.274,111.365,-51.962,-178.769,6.170,148.748
C04302=1183.278,111.116,-51.943,-178.771,6.169,148.748
C04303=1183.284,110.867,-51.925,-178.775,6.168,148.749
C04304=1183.289,110.617,-51.905,-178.777,6.167,148.749
C04305=1183.293,110.369,-51.886,-178.779,6.165,148.750
C04306=1183.299,110.118,-51.867,-178.783,6.164,148.750
C04307=1183.303,109.870,-51.849,-178.785,6.163,148.751
C04308=1183.309,109.620,-51.830,-178.787,6.161,148.751
C04309=1183.313,109.371,-51.811,-178.790,6.160,148.752
C04310=1183.318,109.122,-51.792,-178.793,6.159,148.752
C04311=1183.322,108.872,-51.773,-178.795,6.157,148.753
C04312=1183.327,108.624,-51.755,-178.798,6.156,148.753
C04313=1183.332,108.375,-51.735,-178.801,6.155,148.754
C04314=1183.337,108.125,-51.717,-178.803,6.154,148.754
C04315=1183.342,107.876,-51.698,-178.806,6.152,148.755
C04316=1183.346,107.626,-51.680,-178.809,6.151,148.755
C04317=1183.352,107.377,-51.660,-178.811,6.150,148.756
C04318=1183.357,107.128,-51.642,-178.814,6.148,148.756
C04319=1183.362,106.860,-51.621,-178.817,6.147,148.757
C04320=1183.367,106.591,-51.602,-178.819,6.146,148.757
C04321=1183.372,106.323,-51.581,-178.823,6.145,148.758
C04322=1183.377,106.054,-51.561,-178.825,6.143,148.758
C04323=1183.382,105.805,-51.543,-178.828,6.142,148.759
C04324=1183.387,105.556,-51.524,-178.831,6.141,148.759
C04325=1183.392,105.306,-51.505,-178.833,6.139,148.760
C04326=1183.396,105.058,-51.486,-178.836,6.138,148.760
C04327=1183.401,104.809,-51.468,-178.839,6.137,148.761
C04328=1183.406,104.559,-51.449,-178.841,6.136,148.761
C04329=1183.411,104.310,-51.431,-178.844,6.134,148.762
C04330=1183.416,104.061,-51.411,-178.846,6.133,148.762
C04331=1183.421,103.811,-51.393,-178.849,6.132,148.763
C04332=1183.426,103.562,-51.375,-178.852,6.131,148.763
C04333=1183.431,103.313,-51.356,-178.854,6.129,148.764
C04334=1183.435,103.063,-51.337,-178.857,6.128,148.764
C04335=1183.440,102.814,-51.319,-178.860,6.127,148.765
C04336=1183.445,102.565,-51.301,-178.863,6.126,148.765
C04337=1183.450,102.315,-51.282,-178.865,6.125,148.766
C04338=1183.454,102.067,-51.263,-178.868,6.123,148.766
C04339=1183.459,101.817,-51.245,-178.870,6.122,148.767
C04340=1183.464,101.567,-51.226,-178.873,6.121,148.767
C04341=1183.469,101.318,-51.208,-178.876,6.120,148.768
C04342=1183.474,101.070,-51.190,-178.878,6.118,148.768
C04343=1183.479,100.820,-51.172,-178.881,6.117,148.769
C04344=1183.484,100.570,-51.153,-178.884,6.116,148.769
C04345=1183.489,100.322,-51.134,-178.886,6.114,148.770
C04346=1183.493,100.072,-51.116,-178.889,6.114,148.770
C04347=1183.498,99.823,-51.098,-178.892,6.112,148.771
C04348=1183.503,99.573,-51.079,-178.894,6.112,148.771
C04349=1183.508,99.325,-51.060,-178.897,6.110,148.772
C04350=1183.513,99.075,-51.042,-178.899,6.109,148.772
C04351=1183.518,98.826,-51.024,-178.902,6.108,148.773
C04352=1183.522,98.576,-51.006,-178.904,6.107,148.773
C04353=1183.528,98.327,-50.987,-178.908,6.105,148.774
C04354=1183.532,98.078,-50.969,-178.910,6.104,148.774
C04355=1183.537,97.829,-50.951,-178.912,6.103,148.775
C04356=1183.542,97.579,-50.932,-178.915,6.102,148.775
C04357=1183.547,97.330,-50.914,-178.918,6.100,148.776
C04358=1183.552,97.081,-50.896,-178.920,6.100,148.777
C04359=1183.557,96.831,-50.878,-178.923,6.098,148.777
C04360=1183.562,96.582,-50.860,-178.926,6.098,148.778
C04361=1183.566,96.333,-50.841,-178.928,6.096,148.778
C04362=1183.571,96.084,-50.823,-178.931,6.095,148.778
C04363=1183.576,95.835,-50.805,-178.934,6.094,148.779
C04364=1183.581,95.585,-50.787,-178.936,6.093,148.780
C04365=1183.586,95.336,-50.769,-178.939,6.091,148.780
C04366=1183.591,95.086,-50.750,-178.941,6.090,148.781
C04367=1183.596,94.837,-50.732,-178.944,6.089,148.781
C04368=1183.601,94.588,-50.714,-178.947,6.088,148.782
C04369=1183.605,94.339,-50.696,-178.949,6.086,148.782
C04370=1183.610,94.089,-50.678,-178.952,6.086,148.783
C04371=1183.615,93.840,-50.660,-178.955,6.084,148.783
C04372=1183.620,93.590,-50.642,-178.957,6.084,148.784
C04373=1183.624,93.341,-50.624,-178.960,6.082,148.784
C04374=1183.629,93.092,-50.606,-178.963,6.081,148.785
C04375=1183.634,92.843,-50.588,-178.965,6.080,148.785
C04376=1183.639,92.594,-50.570,-178.968,6.079,148.786
C04377=1183.644,92.344,-50.552,-178.971,6.077,148.786
C04378=1183.649,92.095,-50.534,-178.973,6.076,148.787
C04379=1183.654,91.846,-50.516,-178.976,6.075,148.787
C04380=1183.658,91.596,-50.498,-178.978,6.074,148.788
C04381=1183.663,91.347,-50.480,-178.981,6.073,148.788
C04382=1183.668,91.098,-50.462,-178.983,6.072,148.789
C04383=1183.673,90.849,-50.444,-178.987,6.070,148.789
C04384=1183.678,90.599,-50.426,-178.989,6.070,148.790
C04385=1183.683,90.350,-50.408,-178.992,6.068,148.791
C04386=1183.688,90.101,-50.390,-178.994,6.067,148.791
C04387=1183.693,89.851,-50.372,-178.997,6.066,148.792
C04388=1183.698,89.602,-50.354,-178.999,6.065,148.792
C04389=1183.703,89.353,-50.336,-179.002,6.063,148.792
C04390=1183.708,89.104,-50.318,-179.005,6.063,148.793
C04391=1183.712,88.853,-50.301,-179.008,6.061,148.794
C04392=1183.717,88.604,-50.283,-179.010,6.060,148.794
C04393=1183.722,88.355,-50.265,-179.012,6.060,148.795
C04394=1183.727,88.106,-50.247,-179.016,6.058,148.795
C04395=1183.732,87.857,-50.229,-179.018,6.057,148.796
C04396=1183.737,87.607,-50.212,-179.021,6.056,148.796
C04397=1183.741,87.358,-50.194,-179.023,6.055,148.797
C04398=1183.746,87.109,-50.176,-179.026,6.054,148.797
C04399=1183.751,86.860,-50.158,-179.028,6.053,148.798
C04400=1183.756,86.610,-50.141,-179.032,6.051,148.798
C04401=1183.761,86.361,-50.123,-179.034,6.050,148.799
C04402=1183.766,86.111,-50.105,-179.037,6.049,148.800
C04403=1183.771,85.862,-50.088,-179.039,6.048,148.800
C04404=1183.776,85.612,-50.070,-179.042,6.048,148.801
C04405=1183.781,85.364,-50.052,-179.044,6.046,148.801
C04406=1183.786,85.114,-50.035,-179.046,6.045,148.801
C04407=1183.791,84.865,-50.017,-179.050,6.044,148.802
C04408=1183.796,84.615,-49.999,-179.052,6.043,148.803
C04409=1183.801,84.366,-49.982,-179.055,6.041,148.803
C04410=1183.805,84.117,-49.965,-179.057,6.041,148.804
C04411=1183.810,83.868,-49.947,-179.060,6.039,148.804
C04412=1183.815,83.618,-49.929,-179.063,6.038,148.805
C04413=1183.820,83.369,-49.911,-179.065,6.038,148.805
C04414=1183.825,83.120,-49.893,-179.068,6.036,148.806
C04415=1183.829,82.870,-49.877,-179.070,6.035,148.806
C04416=1183.834,82.621,-49.859,-179.073,6.034,148.807
C04417=1183.840,82.371,-49.841,-179.076,6.033,148.807
C04418=1183.844,82.122,-49.824,-179.078,6.032,148.808
C04419=1183.849,81.872,-49.807,-179.081,6.031,148.809
C04420=1183.854,81.623,-49.789,-179.083,6.030,148.809
C04421=1183.859,81.373,-49.772,-179.087,6.029,148.810
C04422=1183.865,81.125,-49.754,-179.089,6.028,148.810
C04423=1183.870,80.856,-49.735,-179.092,6.026,148.811
C04424=1183.874,80.588,-49.716,-179.095,6.026,148.811
C04425=1183.880,80.319,-49.698,-179.097,6.024,148.812
C04426=1183.885,80.052,-49.679,-179.100,6.023,148.812
C04427=1183.891,79.802,-49.661,-179.103,6.022,148.813
C04428=1183.895,79.552,-49.645,-179.105,6.021,148.814
C04429=1183.900,79.303,-49.627,-179.108,6.020,148.814
C04430=1183.905,79.053,-49.610,-179.111,6.019,148.815
C04431=1183.909,78.805,-49.592,-179.114,6.018,148.815
C04432=1183.915,78.555,-49.575,-179.116,6.017,148.816
C04433=1183.919,78.306,-49.557,-179.119,6.016,148.816
C04434=1183.924,78.056,-49.540,-179.121,6.015,148.817
C04435=1183.930,77.807,-49.523,-179.124,6.014,148.817
C04436=1183.935,77.558,-49.505,-179.127,6.012,148.818
C04437=1183.939,77.308,-49.489,-179.129,6.012,148.818
C04438=1183.944,77.059,-49.471,-179.131,6.011,148.819
C04439=1183.949,76.810,-49.454,-179.135,6.010,148.820
C04440=1183.954,76.560,-49.437,-179.137,6.009,148.820
C04441=1183.959,76.311,-49.419,-179.139,6.008,148.821
C04442=1183.963,76.061,-49.402,-179.142,6.006,148.821
C04443=1183.969,75.812,-49.385,-179.145,6.006,148.822
C04444=1183.973,75.563,-49.368,-179.147,6.004,148.822
C04445=1183.978,75.314,-49.351,-179.150,6.004,148.823
C04446=1183.984,75.064,-49.333,-179.152,6.003,148.823
C04447=1183.988,74.814,-49.317,-179.155,6.001,148.824
C04448=1183.993,74.565,-49.299,-179.158,6.000,148.824
C04449=1183.998,74.316,-49.282,-179.161,5.999,148.825
C04450=1184.003,74.066,-49.265,-179.163,5.998,148.825
C04451=1184.008,73.817,-49.248,-179.166,5.998,148.826
C04452=1184.013,73.568,-49.230,-179.169,5.996,148.827
C04453=1184.017,73.318,-49.214,-179.171,5.995,148.827
C04454=1184.023,73.069,-49.197,-179.174,5.995,148.828
C04455=1184.027,72.820,-49.180,-179.176,5.993,148.828
C04456=1184.032,72.571,-49.162,-179.179,5.993,148.829
C04457=1184.037,72.321,-49.146,-179.181,5.992,148.829
C04458=1184.042,72.071,-49.128,-179.184,5.990,148.830
C04459=1184.047,71.823,-49.112,-179.186,5.990,148.830
C04460=1184.052,71.573,-49.095,-179.190,5.988,148.831
C04461=1184.057,71.323,-49.078,-179.192,5.987,148.831
C04462=1184.062,71.074,-49.060,-179.194,5.987,148.832
C04463=1184.067,70.825,-49.044,-179.197,5.985,148.833
C04464=1184.072,70.575,-49.027,-179.200,5.985,148.833
C04465=1184.077,70.326,-49.010,-179.202,5.984,148.834
C04466=1184.082,70.076,-48.993,-179.205,5.982,148.834
C04467=1184.087,69.827,-48.976,-179.208,5.982,148.835
C04468=1184.092,69.578,-48.959,-179.210,5.981,148.835
C04469=1184.097,69.328,-48.942,-179.213,5.980,148.836
C04470=1184.101,69.079,-48.926,-179.215,5.979,148.837
C04471=1184.107,68.830,-48.909,-179.218,5.978,148.837
C04472=1184.111,68.580,-48.892,-179.221,5.976,148.838
C04473=1184.116,68.331,-48.874,-179.223,5.976,148.838
C04474=1184.121,68.082,-48.858,-179.225,5.975,148.839
C04475=1184.126,67.833,-48.841,-179.229,5.974,148.839
C04476=1184.131,67.583,-48.824,-179.231,5.973,148.840
C04477=1184.135,67.333,-48.807,-179.233,5.972,148.840
C04478=1184.141,67.085,-48.791,-179.237,5.971,148.841
C04479=1184.146,66.835,-48.774,-179.239,5.970,148.842
C04480=1184.150,66.585,-48.757,-179.241,5.969,148.842
C04481=1184.155,66.337,-48.741,-179.244,5.968,148.843
C04482=1184.161,66.086,-48.724,-179.247,5.967,148.843
C04483=1184.165,65.837,-48.707,-179.249,5.967,148.844
C04484=1184.170,65.588,-48.691,-179.252,5.965,148.844
C04485=1184.176,65.338,-48.674,-179.255,5.964,148.845
C04486=1184.180,65.089,-48.657,-179.257,5.964,148.845
C04487=1184.185,64.840,-48.641,-179.260,5.962,148.846
C04488=1184.190,64.590,-48.624,-179.262,5.961,148.847
C04489=1184.195,64.340,-48.607,-179.265,5.961,148.847
C04490=1184.200,64.092,-48.591,-179.267,5.960,148.848
C04491=1184.205,63.842,-48.573,-179.270,5.959,148.848
C04492=1184.210,63.592,-48.557,-179.273,5.958,148.849
C04493=1184.215,63.343,-48.541,-179.275,5.957,148.849
C04494=1184.220,63.094,-48.525,-179.278,5.956,148.850
C04495=1184.225,62.844,-48.508,-179.280,5.955,148.851
C04496=1184.230,62.595,-48.491,-179.283,5.954,148.851
C04497=1184.234,62.345,-48.474,-179.286,5.953,148.852
C04498=1184.239,62.097,-48.458,-179.288,5.952,148.852
C04499=1184.245,61.846,-48.441,-179.291,5.952,148.853
C04500=1184.249,61.597,-48.425,-179.294,5.950,148.853
C04501=1184.254,61.348,-48.408,-179.296,5.949,148.854
C04502=1184.259,61.099,-48.392,-179.298,5.949,148.854
C04503=1184.264,60.849,-48.376,-179.301,5.948,148.855
C04504=1184.270,60.599,-48.359,-179.304,5.947,148.856
C04505=1184.275,60.351,-48.343,-179.306,5.946,148.856
C04506=1184.279,60.101,-48.326,-179.309,5.945,148.857
C04507=1184.284,59.851,-48.310,-179.312,5.944,148.857
C04508=1184.289,59.602,-48.294,-179.314,5.943,148.858
C04509=1184.294,59.352,-48.276,-179.317,5.942,148.858
C04510=1184.299,59.104,-48.260,-179.319,5.942,148.859
C04511=1184.304,58.853,-48.244,-179.322,5.940,148.860
C04512=1184.309,58.605,-48.228,-179.325,5.939,148.860
C04513=1184.314,58.355,-48.211,-179.327,5.939,148.861
C04514=1184.318,58.105,-48.195,-179.329,5.938,148.861
C04515=1184.324,57.856,-48.179,-179.333,5.937,148.862
C04516=1184.329,57.607,-48.162,-179.335,5.936,148.863
C04517=1184.334,57.357,-48.146,-179.337,5.935,148.863
C04518=1184.339,57.108,-48.129,-179.341,5.934,148.864
C04519=1184.344,56.858,-48.114,-179.343,5.933,148.864
C04520=1184.348,56.609,-48.097,-179.345,5.932,148.865
C04521=1184.354,56.360,-48.081,-179.348,5.932,148.866
C04522=1184.358,56.110,-48.065,-179.351,5.930,148.866
C04523=1184.363,55.861,-48.049,-179.353,5.930,148.867
C04524=1184.368,55.611,-48.033,-179.356,5.929,148.867
C04525=1184.373,55.362,-48.016,-179.358,5.928,148.868
C04526=1184.378,55.112,-48.000,-179.361,5.927,148.868
C04527=1184.384,54.844,-47.982,-179.364,5.926,148.869
C04528=1184.390,54.575,-47.965,-179.367,5.925,148.869
C04529=1184.395,54.306,-47.948,-179.369,5.924,148.870
C04530=1184.400,54.038,-47.930,-179.372,5.924,148.871
C04531=1184.405,53.789,-47.914,-179.375,5.922,148.871
C04532=1184.410,53.540,-47.898,-179.377,5.922,148.872
C04533=1184.415,53.290,-47.882,-179.380,5.921,148.873
C04534=1184.420,53.041,-47.865,-179.382,5.920,148.873
C04535=1184.425,52.791,-47.850,-179.385,5.919,148.874
C04536=1184.429,52.542,-47.833,-179.388,5.918,148.874
C04537=1184.435,52.292,-47.818,-179.390,5.917,148.875
C04538=1184.440,52.042,-47.802,-179.393,5.917,148.875
C04539=1184.445,51.793,-47.785,-179.396,5.915,148.876
C04540=1184.450,51.544,-47.770,-179.398,5.915,148.877
C04541=1184.455,51.295,-47.753,-179.400,5.914,148.877
C04542=1184.460,51.045,-47.737,-179.403,5.913,148.878
C04543=1184.464,50.796,-47.721,-179.406,5.912,148.878
C04544=1184.470,50.546,-47.705,-179.408,5.911,148.879
C04545=1184.475,50.296,-47.689,-179.411,5.911,148.879
C04546=1184.479,50.048,-47.674,-179.414,5.910,148.880
C04547=1184.484,49.798,-47.658,-179.416,5.909,148.881
C04548=1184.489,49.548,-47.642,-179.419,5.908,148.881
C04549=1184.494,49.299,-47.626,-179.421,5.907,148.882
C04550=1184.499,49.049,-47.610,-179.424,5.906,148.882
C04551=1184.504,48.800,-47.594,-179.426,5.906,148.883
C04552=1184.509,48.551,-47.578,-179.429,5.904,148.883
C04553=1184.514,48.301,-47.562,-179.432,5.904,148.884
C04554=1184.520,48.052,-47.546,-179.434,5.903,148.885
C04555=1184.524,47.802,-47.530,-179.437,5.902,148.885
C04556=1184.529,47.553,-47.515,-179.439,5.902,148.886
C04557=1184.534,47.304,-47.499,-179.442,5.900,148.886
C04558=1184.539,47.054,-47.483,-179.445,5.900,148.887
C04559=1184.544,46.805,-47.467,-179.447,5.899,148.888
C04560=1184.549,46.555,-47.451,-179.449,5.898,148.888
C04561=1184.554,46.305,-47.435,-179.452,5.898,148.889
C04562=1184.559,46.056,-47.420,-179.455,5.896,148.889
C04563=1184.564,45.807,-47.404,-179.457,5.895,148.890
C04564=1184.569,45.557,-47.388,-179.460,5.895,148.891
C04565=1184.574,45.308,-47.372,-179.462,5.894,148.891
C04566=1184.579,45.058,-47.357,-179.465,5.894,148.892
C04567=1184.584,44.808,-47.341,-179.468,5.892,148.892
C04568=1184.589,44.560,-47.325,-179.470,5.891,148.893
C04569=1184.594,44.311,-47.310,-179.473,5.891,148.893
C04570=1184.599,44.060,-47.294,-179.476,5.890,148.894
C04571=1184.604,43.811,-47.278,-179.478,5.889,148.895
C04572=1184.609,43.562,-47.263,-179.481,5.888,148.895
C04573=1184.614,43.312,-47.247,-179.484,5.888,148.896
C04574=1184.619,43.062,-47.232,-179.486,5.887,148.896
C04575=1184.624,42.814,-47.215,-179.488,5.886,148.897
C04576=1184.628,42.564,-47.200,-179.490,5.885,148.897
C04577=1184.633,42.314,-47.184,-179.494,5.884,148.898
C04578=1184.639,42.065,-47.169,-179.496,5.884,148.899
C04579=1184.644,41.816,-47.153,-179.498,5.883,148.899
C04580=1184.648,41.566,-47.138,-179.501,5.882,148.900
C04581=1184.654,41.316,-47.122,-179.504,5.882,148.901
C04582=1184.659,41.067,-47.107,-179.506,5.881,148.901
C04583=1184.664,40.818,-47.091,-179.509,5.879,148.902
C04584=1184.669,40.568,-47.076,-179.512,5.879,148.902
C04585=1184.674,40.318,-47.060,-179.514,5.878,148.903
C04586=1184.679,40.069,-47.044,-179.517,5.878,148.904
C04587=1184.684,39.820,-47.029,-179.519,5.877,148.904
C04588=1184.689,39.570,-47.014,-179.521,5.876,148.905
C04589=1184.694,39.320,-46.998,-179.525,5.875,148.905
C04590=1184.699,39.071,-46.983,-179.527,5.874,148.906
C04591=1184.704,38.822,-46.967,-179.529,5.873,148.906
C04592=1184.709,38.572,-46.951,-179.532,5.873,148.907
C04593=1184.714,38.323,-46.936,-179.534,5.872,148.908
C04594=1184.719,38.073,-46.921,-179.537,5.872,148.908
C04595=1184.724,37.824,-46.906,-179.540,5.870,148.909
C04596=1184.729,37.575,-46.890,-179.542,5.869,148.909
C04597=1184.734,37.325,-46.874,-179.545,5.869,148.910
C04598=1184.738,37.076,-46.859,-179.548,5.868,148.911
C04599=1184.744,36.826,-46.844,-179.550,5.868,148.911
C04600=1184.750,36.576,-46.829,-179.552,5.867,148.912
C04601=1184.754,36.327,-46.814,-179.556,5.866,148.912
C04602=1184.760,36.078,-46.798,-179.558,5.865,148.913
C04603=1184.764,35.828,-46.783,-179.560,5.864,148.914
C04604=1184.769,35.579,-46.767,-179.563,5.864,148.914
C04605=1184.774,35.329,-46.752,-179.565,5.863,148.915
C04606=1184.779,35.080,-46.737,-179.568,5.862,148.915
C04607=1184.785,34.830,-46.722,-179.570,5.862,148.916
C04608=1184.789,34.580,-46.706,-179.573,5.860,148.917
C04609=1184.794,34.331,-46.691,-179.576,5.860,148.917
C04610=1184.799,34.082,-46.676,-179.578,5.859,148.918
C04611=1184.804,33.832,-46.660,-179.581,5.858,148.918
C04612=1184.809,33.583,-46.646,-179.583,5.858,148.919
C04613=1184.815,33.333,-46.630,-179.586,5.857,148.920
C04614=1184.819,33.084,-46.615,-179.588,5.857,148.920
C04615=1184.824,32.834,-46.599,-179.591,5.856,148.921
C04616=1184.829,32.585,-46.585,-179.594,5.855,148.921
C04617=1184.834,32.335,-46.570,-179.596,5.854,148.922
C04618=1184.839,32.086,-46.555,-179.599,5.853,148.923
C04619=1184.844,31.836,-46.539,-179.601,5.853,148.923
C04620=1184.849,31.587,-46.525,-179.604,5.852,148.924
C04621=1184.855,31.337,-46.509,-179.606,5.851,148.924
C04622=1184.859,31.088,-46.494,-179.609,5.851,148.925
C04623=1184.865,30.839,-46.479,-179.611,5.850,148.926
C04624=1184.869,30.588,-46.464,-179.614,5.849,148.926
C04625=1184.874,30.339,-46.449,-179.617,5.848,148.927
C04626=1184.879,30.090,-46.433,-179.619,5.847,148.927
C04627=1184.884,29.840,-46.419,-179.622,5.847,148.928
C04628=1184.889,29.591,-46.404,-179.624,5.846,148.929
C04629=1184.894,29.342,-46.389,-179.626,5.846,148.929
C04630=1184.900,29.092,-46.374,-179.629,5.845,148.930
C04631=1184.905,28.823,-46.358,-179.632,5.844,148.931
C04632=1184.910,28.554,-46.341,-179.635,5.843,148.931
C04633=1184.916,28.286,-46.325,-179.638,5.843,148.932
C04634=1184.921,28.017,-46.309,-179.640,5.842,148.933
C04635=1184.926,27.767,-46.294,-179.642,5.841,148.933
C04636=1184.931,27.518,-46.280,-179.646,5.840,148.934
C04637=1184.936,27.268,-46.264,-179.648,5.840,148.934
C04638=1184.941,27.019,-46.250,-179.650,5.839,148.935
C04639=1184.946,26.770,-46.235,-179.653,5.838,148.935
C04640=1184.952,26.519,-46.220,-179.656,5.838,148.936
C04641=1184.956,26.270,-46.205,-179.658,5.837,148.937
C04642=1184.961,26.021,-46.191,-179.661,5.836,148.937
C04643=1184.967,25.771,-46.175,-179.663,5.836,148.938
C04644=1184.972,25.522,-46.161,-179.665,5.835,148.938
C04645=1184.976,25.272,-46.146,-179.668,5.834,148.939
C04646=1184.982,25.022,-46.131,-179.671,5.834,148.940
C04647=1184.987,24.773,-46.116,-179.673,5.832,148.940
C04648=1184.992,24.524,-46.102,-179.676,5.832,148.941
C04649=1184.997,24.274,-46.086,-179.679,5.831,148.942
C04650=1185.002,24.025,-46.072,-179.681,5.831,148.942
C04651=1185.007,23.775,-46.057,-179.684,5.830,148.943
C04652=1185.012,23.526,-46.043,-179.686,5.829,148.943
C04653=1185.017,23.276,-46.027,-179.689,5.829,148.944
C04654=1185.022,23.027,-46.013,-179.691,5.828,148.945
C04655=1185.027,22.777,-45.998,-179.694,5.828,148.945
C04656=1185.032,22.528,-45.983,-179.696,5.827,148.946
C04657=1185.037,22.278,-45.969,-179.698,5.826,148.946
C04658=1185.042,22.029,-45.954,-179.701,5.826,148.947
C04659=1185.047,21.779,-45.939,-179.704,5.825,148.948
C04660=1185.052,21.529,-45.925,-179.706,5.824,148.948
C04661=1185.057,21.280,-45.909,-179.709,5.823,148.949
C04662=1185.062,21.030,-45.895,-179.712,5.823,148.950
C04663=1185.067,20.780,-45.881,-179.714,5.822,148.950
C04664=1185.072,20.531,-45.866,-179.717,5.821,148.951
C04665=1185.077,20.281,-45.851,-179.719,5.821,148.951
C04666=1185.082,20.032,-45.837,-179.722,5.820,148.952
C04667=1185.087,19.783,-45.822,-179.724,5.819,148.952
C04668=1185.093,19.534,-45.808,-179.727,5.819,148.953
C04669=1185.098,19.284,-45.793,-179.729,5.818,148.954
C04670=1185.102,19.035,-45.779,-179.731,5.818,148.954
C04671=1185.108,18.785,-45.764,-179.734,5.817,148.955
C04672=1185.113,18.535,-45.749,-179.737,5.817,148.956
C04673=1185.118,18.285,-45.735,-179.739,5.816,148.956
C04674=1185.122,18.036,-45.720,-179.742,5.815,148.957
C04675=1185.127,17.787,-45.706,-179.744,5.815,148.957
C04676=1185.132,17.537,-45.692,-179.747,5.814,148.958
C04677=1185.137,17.287,-45.677,-179.749,5.813,148.959
C04678=1185.143,17.038,-45.662,-179.752,5.812,148.959
C04679=1185.148,16.789,-45.648,-179.755,5.812,148.960
C04680=1185.153,16.539,-45.633,-179.757,5.811,148.960
C04681=1185.158,16.289,-45.619,-179.760,5.810,148.961
C04682=1185.163,16.040,-45.605,-179.762,5.810,148.962
C04683=1185.168,15.790,-45.590,-179.765,5.809,148.962
C04684=1185.173,15.541,-45.576,-179.767,5.808,148.963
C04685=1185.178,15.292,-45.562,-179.770,5.808,148.964
C04686=1185.183,15.042,-45.547,-179.773,5.807,148.964
C04687=1185.188,14.792,-45.533,-179.775,5.807,148.965
C04688=1185.194,14.542,-45.518,-179.777,5.806,148.965
C04689=1185.199,14.293,-45.504,-179.780,5.806,148.966
C04690=1185.203,14.043,-45.489,-179.782,5.805,148.967
C04691=1185.208,13.794,-45.475,-179.785,5.804,148.967
C04692=1185.214,13.545,-45.461,-179.787,5.804,148.968
C04693=1185.219,13.295,-45.447,-179.790,5.803,148.969
C04694=1185.224,13.045,-45.432,-179.792,5.802,148.969
C04695=1185.229,12.796,-45.418,-179.795,5.802,148.970
C04696=1185.234,12.546,-45.404,-179.798,5.801,148.970
C04697=1185.239,12.297,-45.390,-179.800,5.801,148.971
C04698=1185.244,12.047,-45.376,-179.802,5.800,148.972
C04699=1185.249,11.797,-45.361,-179.805,5.800,148.972
C04700=1185.254,11.548,-45.347,-179.807,5.799,148.973
C04701=1185.259,11.298,-45.333,-179.810,5.798,148.973
C04702=1185.265,11.049,-45.319,-179.812,5.798,148.974
C04703=1185.270,10.799,-45.305,-179.815,5.797,148.975
C04704=1185.275,10.550,-45.290,-179.817,5.796,148.975
C04705=1185.280,10.300,-45.276,-179.820,5.796,148.976
C04706=1185.285,10.051,-45.262,-179.823,5.796,148.977
C04707=1185.290,9.801,-45.248,-179.825,5.795,148.977
C04708=1185.295,9.552,-45.234,-179.827,5.794,148.978
C04709=1185.300,9.302,-45.219,-179.830,5.794,148.978
C04710=1185.304,9.052,-45.206,-179.833,5.793,148.979
C04711=1185.310,8.803,-45.192,-179.835,5.792,148.980
C04712=1185.315,8.554,-45.177,-179.838,5.792,148.980
C04713=1185.320,8.304,-45.163,-179.840,5.791,148.981
C04714=1185.325,8.054,-45.149,-179.842,5.791,148.981
C04715=1185.330,7.805,-45.135,-179.845,5.790,148.982
C04716=1185.335,7.556,-45.121,-179.848,5.790,148.983
C04717=1185.340,7.306,-45.106,-179.850,5.789,148.983
C04718=1185.346,7.056,-45.093,-179.852,5.788,148.984
C04719=1185.351,6.806,-45.079,-179.855,5.788,148.985
C04720=1185.355,6.557,-45.065,-179.858,5.787,148.985
C04721=1185.360,6.307,-45.051,-179.860,5.787,148.986
C04722=1185.366,6.058,-45.037,-179.863,5.786,148.986
C04723=1185.371,5.809,-45.023,-179.865,5.785,148.987
C04724=1185.376,5.559,-45.008,-179.868,5.785,148.988
C04725=1185.381,5.309,-44.995,-179.870,5.784,148.988
C04726=1185.386,5.060,-44.981,-179.873,5.784,148.989
C04727=1185.391,4.810,-44.967,-179.875,5.783,148.990
C04728=1185.396,4.561,-44.953,-179.878,5.783,148.990
C04729=1185.401,4.311,-44.939,-179.880,5.782,148.991
C04730=1185.406,4.061,-44.926,-179.883,5.781,148.991
C04731=1185.411,3.811,-44.911,-179.886,5.781,148.992
C04732=1185.417,3.562,-44.897,-179.888,5.780,148.993
C04733=1185.421,3.313,-44.884,-179.890,5.780,148.993
C04734=1185.426,3.063,-44.870,-179.893,5.779,148.994
C04735=1185.432,2.795,-44.855,-179.896,5.779,148.995
C04736=1185.438,2.525,-44.840,-179.898,5.778,148.995
C04737=1185.443,2.256,-44.825,-179.901,5.778,148.996
C04738=1185.448,1.986,-44.810,-179.904,5.777,148.997
C04739=1185.454,1.737,-44.797,-179.906,5.776,148.997
C04740=1185.458,1.487,-44.783,-179.908,5.776,148.998
C04741=1185.463,1.238,-44.769,-179.911,5.775,148.999
C04742=1185.469,0.989,-44.755,-179.914,5.775,148.999
C04743=1185.474,0.738,-44.741,-179.916,5.774,149.000
C04744=1185.479,0.490,-44.728,-179.919,5.774,149.000
C04745=1185.484,0.240,-44.714,-179.921,5.773,149.001
C04746=1185.489,-0.010,-44.700,-179.923,5.772,149.002
C04747=1185.494,-0.259,-44.687,-179.926,5.772,149.002
C04748=1185.499,-0.509,-44.673,-179.929,5.771,149.003
C04749=1185.505,-0.758,-44.659,-179.931,5.771,149.004
C04750=1185.510,-1.008,-44.645,-179.934,5.770,149.004
C04751=1185.514,-1.258,-44.632,-179.936,5.769,149.005
C04752=1185.520,-1.507,-44.618,-179.939,5.769,149.005
C04753=1185.525,-1.757,-44.604,-179.941,5.768,149.006
C04754=1185.530,-2.006,-44.591,-179.944,5.768,149.007
C04755=1185.535,-2.256,-44.577,-179.946,5.767,149.007
C04756=1185.540,-2.506,-44.563,-179.949,5.767,149.008
C04757=1185.545,-2.755,-44.550,-179.951,5.767,149.008
C04758=1185.550,-3.005,-44.536,-179.953,5.766,149.009
C04759=1185.556,-3.254,-44.523,-179.956,5.766,149.010
C04760=1185.560,-3.504,-44.510,-179.958,5.765,149.011
C04761=1185.566,-3.753,-44.496,-179.961,5.764,149.011
C04762=1185.571,-4.004,-44.482,-179.963,5.764,149.012
C04763=1185.575,-4.253,-44.468,-179.966,5.763,149.012
C04764=1185.581,-4.502,-44.455,-179.969,5.763,149.013
C04765=1185.586,-4.752,-44.442,-179.971,5.762,149.014
C04766=1185.591,-5.002,-44.428,-179.973,5.762,149.014
C04767=1185.596,-5.251,-44.414,-179.976,5.761,149.015
C04768=1185.601,-5.501,-44.401,-179.978,5.760,149.015
C04769=1185.606,-5.750,-44.387,-179.981,5.760,149.016
C04770=1185.612,-6.000,-44.375,-179.984,5.759,149.017
C04771=1185.616,-6.250,-44.360,-179.986,5.759,149.017
C04772=1185.622,-6.499,-44.347,-179.988,5.759,149.018
C04773=1185.627,-6.749,-44.333,-179.990,5.758,149.019
C04774=1185.632,-6.998,-44.320,-179.993,5.758,149.019
C04775=1185.637,-7.248,-44.307,-179.996,5.758,149.020
C04776=1185.643,-7.497,-44.293,-179.998,5.757,149.020
C04777=1185.647,-7.747,-44.280,179.999,5.756,149.021
C04778=1185.653,-7.996,-44.267,179.997,5.756,149.022
C04779=1185.657,-8.246,-44.254,179.995,5.755,149.022
C04780=1185.663,-8.496,-44.240,179.992,5.754,149.023
C04781=1185.667,-8.745,-44.227,179.989,5.754,149.024
C04782=1185.673,-8.995,-44.213,179.987,5.753,149.024
C04783=1185.677,-9.244,-44.200,179.984,5.753,149.025
C04784=1185.683,-9.494,-44.187,179.982,5.753,149.026
C04785=1185.688,-9.744,-44.174,179.980,5.753,149.026
C04786=1185.693,-9.993,-44.160,179.977,5.752,149.027
C04787=1185.698,-10.243,-44.147,179.975,5.751,149.027
C04788=1185.704,-10.493,-44.134,179.972,5.751,149.028
C04789=1185.708,-10.742,-44.120,179.970,5.750,149.029
C04790=1185.714,-10.992,-44.107,179.967,5.750,149.029
C04791=1185.719,-11.241,-44.094,179.965,5.749,149.030
C04792=1185.724,-11.491,-44.081,179.962,5.748,149.031
C04793=1185.729,-11.740,-44.067,179.959,5.748,149.031
C04794=1185.734,-11.990,-44.054,179.958,5.748,149.032
C04795=1185.739,-12.240,-44.041,179.955,5.748,149.032
C04796=1185.745,-12.490,-44.027,179.952,5.747,149.033
C04797=1185.749,-12.739,-44.014,179.950,5.747,149.034
C04798=1185.754,-12.988,-44.002,179.948,5.746,149.034
C04799=1185.760,-13.238,-43.988,179.945,5.745,149.035
C04800=1185.765,-13.488,-43.975,179.942,5.745,149.036
C04801=1185.770,-13.737,-43.961,179.940,5.744,149.036
C04802=1185.775,-13.987,-43.949,179.938,5.744,149.037
C04803=1185.779,-14.237,-43.936,179.935,5.743,149.038
C04804=1185.785,-14.486,-43.922,179.933,5.743,149.038
C04805=1185.790,-14.736,-43.910,179.930,5.743,149.039
C04806=1185.796,-14.986,-43.896,179.928,5.742,149.039
C04807=1185.801,-15.235,-43.883,179.925,5.742,149.040
C04808=1185.806,-15.484,-43.870,179.923,5.741,149.041
C04809=1185.811,-15.734,-43.857,179.920,5.741,149.041
C04810=1185.816,-15.984,-43.844,179.918,5.740,149.042
C04811=1185.821,-16.234,-43.831,179.915,5.739,149.043
C04812=1185.826,-16.483,-43.818,179.913,5.740,149.043
C04813=1185.832,-16.733,-43.805,179.911,5.739,149.044
C04814=1185.836,-16.982,-43.791,179.908,5.738,149.044
C04815=1185.842,-17.232,-43.778,179.906,5.738,149.045
C04816=1185.847,-17.481,-43.766,179.903,5.738,149.046
C04817=1185.851,-17.731,-43.753,179.901,5.737,149.046
C04818=1185.857,-17.981,-43.740,179.898,5.736,149.047
C04819=1185.862,-18.230,-43.727,179.895,5.736,149.048
C04820=1185.867,-18.480,-43.714,179.893,5.736,149.048
C04821=1185.873,-18.730,-43.701,179.891,5.735,149.049
C04822=1185.878,-18.979,-43.688,179.889,5.735,149.050
C04823=1185.882,-19.229,-43.675,179.886,5.734,149.050
C04824=1185.888,-19.478,-43.662,179.883,5.734,149.051
C04825=1185.893,-19.728,-43.650,179.881,5.733,149.051
C04826=1185.898,-19.978,-43.637,179.878,5.733,149.052
C04827=1185.903,-20.227,-43.624,179.876,5.733,149.053
C04828=1185.909,-20.477,-43.611,179.874,5.732,149.054
C04829=1185.913,-20.727,-43.598,179.871,5.732,149.054
C04830=1185.918,-20.976,-43.585,179.869,5.731,149.055
C04831=1185.924,-21.225,-43.573,179.866,5.731,149.055
C04832=1185.929,-21.475,-43.559,179.864,5.730,149.056
C04833=1185.934,-21.725,-43.546,179.861,5.729,149.057
C04834=1185.939,-21.974,-43.534,179.859,5.730,149.057
C04835=1185.944,-22.224,-43.521,179.857,5.729,149.058
C04836=1185.949,-22.474,-43.508,179.854,5.728,149.058
C04837=1185.955,-22.723,-43.495,179.852,5.728,149.059
C04838=1185.960,-22.973,-43.483,179.849,5.728,149.060
C04839=1185.965,-23.243,-43.468,179.846,5.727,149.061
C04840=1185.971,-23.512,-43.455,179.844,5.727,149.061
C04841=1185.976,-23.782,-43.442,179.841,5.726,149.062
C04842=1185.982,-24.052,-43.428,179.838,5.726,149.063
C04843=1185.987,-24.301,-43.415,179.836,5.725,149.063
C04844=1185.992,-24.551,-43.402,179.834,5.725,149.064
C04845=1185.997,-24.800,-43.390,179.832,5.725,149.064
C04846=1186.002,-25.050,-43.377,179.829,5.724,149.065
C04847=1186.008,-25.300,-43.364,179.827,5.724,149.066
C04848=1186.013,-25.550,-43.352,179.824,5.723,149.066
C04849=1186.018,-25.799,-43.339,179.821,5.723,149.067
C04850=1186.023,-26.049,-43.326,179.819,5.723,149.068
C04851=1186.028,-26.298,-43.314,179.817,5.722,149.068
C04852=1186.033,-26.548,-43.301,179.814,5.722,149.069
C04853=1186.038,-26.797,-43.288,179.812,5.721,149.070
C04854=1186.043,-27.048,-43.276,179.809,5.721,149.070
C04855=1186.049,-27.297,-43.263,179.807,5.720,149.071
C04856=1186.054,-27.547,-43.250,179.805,5.720,149.071
C04857=1186.059,-27.796,-43.238,179.802,5.720,149.072
C04858=1186.065,-28.046,-43.226,179.800,5.719,149.073
C04859=1186.069,-28.296,-43.213,179.797,5.719,149.073
C04860=1186.074,-28.545,-43.200,179.795,5.718,149.074
C04861=1186.079,-28.794,-43.188,179.793,5.718,149.075
C04862=1186.085,-29.044,-43.176,179.790,5.718,149.075
C04863=1186.090,-29.294,-43.163,179.788,5.717,149.076
C04864=1186.095,-29.543,-43.151,179.785,5.717,149.077
C04865=1186.100,-29.793,-43.138,179.783,5.716,149.077
C04866=1186.105,-30.043,-43.126,179.780,5.715,149.078
C04867=1186.110,-30.292,-43.113,179.778,5.716,149.078
C04868=1186.115,-30.542,-43.101,179.776,5.715,149.079
C04869=1186.121,-30.792,-43.089,179.773,5.715,149.080
C04870=1186.126,-31.041,-43.076,179.771,5.714,149.080
C04871=1186.130,-31.291,-43.063,179.768,5.714,149.081
C04872=1186.136,-31.541,-43.051,179.766,5.714,149.082
C04873=1186.142,-31.790,-43.038,179.763,5.714,149.082
C04874=1186.147,-32.040,-43.025,179.761,5.713,149.083
C04875=1186.152,-32.290,-43.014,179.759,5.712,149.084
C04876=1186.157,-32.539,-43.002,179.756,5.712,149.084
C04877=1186.162,-32.789,-42.990,179.754,5.712,149.085
C04878=1186.167,-33.038,-42.977,179.752,5.711,149.085
C04879=1186.172,-33.288,-42.964,179.749,5.711,149.086
C04880=1186.177,-33.538,-42.952,179.746,5.710,149.087
C04881=1186.182,-33.787,-42.940,179.744,5.710,149.087
C04882=1186.188,-34.037,-42.928,179.742,5.710,149.088
C04883=1186.193,-34.286,-42.915,179.739,5.709,149.089
C04884=1186.198,-34.536,-42.903,179.737,5.709,149.089
C04885=1186.203,-34.786,-42.891,179.735,5.708,149.090
C04886=1186.208,-35.035,-42.878,179.732,5.708,149.091
C04887=1186.214,-35.285,-42.866,179.730,5.708,149.091
C04888=1186.219,-35.534,-42.854,179.727,5.708,149.092
C04889=1186.224,-35.785,-42.841,179.725,5.707,149.092
C04890=1186.229,-36.034,-42.829,179.722,5.706,149.093
C04891=1186.234,-36.284,-42.817,179.720,5.706,149.094
C04892=1186.239,-36.534,-42.804,179.718,5.706,149.095
C04893=1186.245,-36.783,-42.792,179.715,5.705,149.095
C04894=1186.250,-37.033,-42.780,179.713,5.705,149.096
C04895=1186.255,-37.282,-42.768,179.710,5.705,149.096
C04896=1186.260,-37.532,-42.756,179.708,5.705,149.097
C04897=1186.265,-37.782,-42.744,179.706,5.704,149.098
C04898=1186.270,-38.031,-42.731,179.703,5.704,149.098
C04899=1186.276,-38.281,-42.720,179.700,5.703,149.099
C04900=1186.281,-38.531,-42.708,179.698,5.702,149.099
C04901=1186.286,-38.780,-42.695,179.696,5.703,149.100
C04902=1186.292,-39.030,-42.683,179.694,5.702,149.101
C04903=1186.296,-39.279,-42.671,179.691,5.702,149.102
C04904=1186.302,-39.529,-42.659,179.689,5.701,149.102
C04905=1186.307,-39.779,-42.647,179.687,5.701,149.103
C04906=1186.312,-40.028,-42.635,179.684,5.701,149.103
C04907=1186.318,-40.278,-42.623,179.681,5.701,149.104
C04908=1186.323,-40.528,-42.610,179.679,5.700,149.105
C04909=1186.327,-40.777,-42.599,179.677,5.700,149.105
C04910=1186.333,-41.027,-42.587,179.674,5.700,149.106
C04911=1186.338,-41.276,-42.575,179.672,5.699,149.106
C04912=1186.343,-41.526,-42.563,179.670,5.698,149.107
C04913=1186.349,-41.776,-42.551,179.667,5.698,149.108
C04914=1186.353,-42.025,-42.539,179.665,5.698,149.109
C04915=1186.359,-42.275,-42.527,179.663,5.697,149.109
C04916=1186.364,-42.525,-42.515,179.660,5.697,149.110
C04917=1186.369,-42.774,-42.502,179.657,5.697,149.110
C04918=1186.374,-43.024,-42.491,179.655,5.697,149.111
C04919=1186.379,-43.274,-42.479,179.653,5.696,149.112
C04920=1186.384,-43.523,-42.467,179.650,5.696,149.112
C04921=1186.390,-43.773,-42.455,179.648,5.695,149.113
C04922=1186.395,-44.023,-42.443,179.646,5.695,149.113
C04923=1186.400,-44.273,-42.432,179.643,5.695,149.114
C04924=1186.405,-44.522,-42.419,179.641,5.694,149.115
C04925=1186.411,-44.772,-42.407,179.638,5.694,149.116
C04926=1186.415,-45.022,-42.396,179.637,5.694,149.116
C04927=1186.421,-45.272,-42.384,179.634,5.693,149.117
C04928=1186.426,-45.521,-42.371,179.631,5.693,149.117
C04929=1186.431,-45.771,-42.360,179.629,5.693,149.118
C04930=1186.436,-46.021,-42.348,179.627,5.693,149.119
C04931=1186.441,-46.271,-42.336,179.624,5.692,149.119
C04932=1186.447,-46.520,-42.324,179.622,5.692,149.120
C04933=1186.452,-46.769,-42.313,179.619,5.691,149.121
C04934=1186.457,-47.019,-42.301,179.617,5.691,149.121
C04935=1186.463,-47.269,-42.289,179.615,5.691,149.122
C04936=1186.467,-47.518,-42.278,179.612,5.690,149.123
C04937=1186.473,-47.768,-42.266,179.610,5.690,149.123
C04938=1186.478,-48.018,-42.254,179.608,5.690,149.124
C04939=1186.483,-48.267,-42.242,179.605,5.689,149.125
C04940=1186.488,-48.517,-42.230,179.603,5.689,149.125
C04941=1186.493,-48.767,-42.218,179.601,5.689,149.126
C04942=1186.498,-49.017,-42.207,179.598,5.689,149.126
C04943=1186.504,-49.286,-42.194,179.595,5.688,149.127
C04944=1186.509,-49.557,-42.181,179.593,5.688,149.128
C04945=1186.515,-49.828,-42.169,179.590,5.687,149.128
C04946=1186.521,-50.097,-42.156,179.587,5.687,149.129
C04947=1186.526,-50.347,-42.144,179.586,5.687,149.130
C04948=1186.532,-50.597,-42.133,179.583,5.686,149.130
C04949=1186.536,-50.847,-42.121,179.581,5.686,149.131
C04950=1186.542,-51.097,-42.109,179.578,5.685,149.132
C04951=1186.547,-51.346,-42.098,179.576,5.685,149.132
C04952=1186.553,-51.596,-42.087,179.574,5.685,149.133
C04953=1186.557,-51.845,-42.075,179.571,5.685,149.134
C04954=1186.563,-52.095,-42.063,179.569,5.685,149.134
C04955=1186.568,-52.345,-42.052,179.567,5.684,149.135
C04956=1186.573,-52.595,-42.040,179.564,5.684,149.136
C04957=1186.578,-52.844,-42.028,179.561,5.683,149.136
C04958=1186.583,-53.093,-42.017,179.560,5.683,149.137
C04959=1186.589,-53.343,-42.005,179.557,5.683,149.137
C04960=1186.594,-53.593,-41.994,179.554,5.682,149.138
C04961=1186.599,-53.843,-41.982,179.553,5.682,149.139
C04962=1186.604,-54.093,-41.971,179.550,5.682,149.139
C04963=1186.609,-54.343,-41.959,179.548,5.682,149.140
C04964=1186.615,-54.592,-41.948,179.545,5.681,149.141
C04965=1186.620,-54.841,-41.936,179.543,5.681,149.141
C04966=1186.625,-55.091,-41.925,179.541,5.681,149.142
C04967=1186.630,-55.341,-41.913,179.538,5.680,149.143
C04968=1186.635,-55.591,-41.902,179.536,5.680,149.143
C04969=1186.641,-55.840,-41.890,179.534,5.680,149.144
C04970=1186.645,-56.090,-41.879,179.531,5.679,149.144
C04971=1186.651,-56.339,-41.867,179.529,5.680,149.145
C04972=1186.656,-56.589,-41.856,179.527,5.679,149.146
C04973=1186.661,-56.839,-41.844,179.524,5.678,149.146
C04974=1186.666,-57.088,-41.833,179.521,5.678,149.147
C04975=1186.672,-57.339,-41.822,179.520,5.678,149.148
C04976=1186.677,-57.588,-41.811,179.517,5.678,149.148
C04977=1186.682,-57.838,-41.799,179.514,5.677,149.149
C04978=1186.687,-58.087,-41.788,179.512,5.678,149.150
C04979=1186.692,-58.337,-41.777,179.510,5.677,149.150
C04980=1186.698,-58.587,-41.765,179.508,5.676,149.151
C04981=1186.702,-58.836,-41.753,179.505,5.677,149.152
C04982=1186.709,-59.086,-41.743,179.503,5.676,149.152
C04983=1186.713,-59.336,-41.731,179.501,5.675,149.153
C04984=1186.719,-59.586,-41.719,179.499,5.676,149.153
C04985=1186.723,-59.835,-41.708,179.496,5.675,149.154
C04986=1186.729,-60.084,-41.697,179.494,5.675,149.155
C04987=1186.734,-60.334,-41.685,179.491,5.674,149.155
C04988=1186.739,-60.584,-41.675,179.489,5.674,149.156
C04989=1186.744,-60.834,-41.663,179.487,5.674,149.157
C04990=1186.750,-61.083,-41.652,179.484,5.673,149.157
C04991=1186.755,-61.333,-41.641,179.482,5.674,149.158
C04992=1186.760,-61.583,-41.629,179.480,5.673,149.158
C04993=1186.765,-61.833,-41.618,179.477,5.672,149.159
C04994=1186.770,-62.082,-41.607,179.475,5.673,149.160
C04995=1186.776,-62.332,-41.595,179.472,5.672,149.161
C04996=1186.781,-62.582,-41.585,179.470,5.672,149.161
C04997=1186.786,-62.831,-41.574,179.468,5.672,149.162
C04998=1186.791,-63.081,-41.562,179.465,5.671,149.162
C04999=1186.796,-63.331,-41.551,179.463,5.671,149.163
C05000=1186.802,-63.580,-41.541,179.461,5.671,149.164
C05001=1186.807,-63.830,-41.529,179.459,5.671,149.164
C05002=1186.812,-64.080,-41.517,179.456,5.670,149.165
C05003=1186.817,-64.329,-41.507,179.454,5.670,149.165
C05004=1186.823,-64.579,-41.495,179.452,5.670,149.166
C05005=1186.828,-64.829,-41.484,179.449,5.669,149.167
C05006=1186.833,-65.078,-41.474,179.447,5.669,149.167
C05007=1186.839,-65.328,-41.462,179.445,5.669,149.168
C05008=1186.844,-65.579,-41.451,179.442,5.668,149.169
C05009=1186.849,-65.827,-41.440,179.440,5.668,149.169
C05010=1186.854,-66.077,-41.429,179.438,5.668,149.170
C05011=1186.859,-66.328,-41.418,179.435,5.668,149.171
C05012=1186.865,-66.577,-41.407,179.433,5.668,149.171
C05013=1186.869,-66.826,-41.396,179.431,5.667,149.172
C05014=1186.874,-67.076,-41.385,179.428,5.667,149.173
C05015=1186.880,-67.326,-41.374,179.427,5.667,149.173
C05016=1186.885,-67.576,-41.363,179.424,5.666,149.174
C05017=1186.890,-67.826,-41.352,179.421,5.666,149.174
C05018=1186.896,-68.075,-41.342,179.419,5.666,149.175
C05019=1186.901,-68.325,-41.330,179.417,5.665,149.176
C05020=1186.906,-68.574,-41.319,179.414,5.665,149.176
C05021=1186.911,-68.824,-41.308,179.412,5.665,149.177
C05022=1186.916,-69.074,-41.297,179.410,5.665,149.178
C05023=1186.922,-69.324,-41.286,179.407,5.664,149.178
C05024=1186.927,-69.573,-41.275,179.405,5.665,149.179
C05025=1186.933,-69.823,-41.265,179.403,5.664,149.179
C05026=1186.937,-70.072,-41.253,179.400,5.663,149.180
C05027=1186.942,-70.323,-41.243,179.398,5.664,149.181
C05028=1186.948,-70.572,-41.231,179.396,5.663,149.181
C05029=1186.953,-70.822,-41.221,179.394,5.663,149.182
C05030=1186.959,-71.071,-41.210,179.391,5.663,149.183
C05031=1186.964,-71.321,-41.199,179.389,5.662,149.183
C05032=1186.968,-71.571,-41.188,179.387,5.662,149.184
C05033=1186.975,-71.821,-41.177,179.384,5.662,149.185
C05034=1186.979,-72.070,-41.166,179.382,5.661,149.185
C05035=1186.985,-72.320,-41.155,179.380,5.662,149.186
C05036=1186.990,-72.570,-41.145,179.378,5.661,149.187
C05037=1186.995,-72.819,-41.134,179.375,5.661,149.187
C05038=1187.000,-73.069,-41.123,179.373,5.661,149.188
C05039=1187.006,-73.318,-41.112,179.371,5.660,149.188
C05040=1187.011,-73.569,-41.101,179.368,5.660,149.189
C05041=1187.017,-73.818,-41.090,179.366,5.660,149.190
C05042=1187.022,-74.068,-41.080,179.364,5.660,149.190
C05043=1187.027,-74.318,-41.069,179.362,5.660,149.191
C05044=1187.032,-74.567,-41.058,179.359,5.659,149.192
C05045=1187.037,-74.817,-41.048,179.357,5.659,149.192
C05046=1187.042,-75.067,-41.038,179.355,5.659,149.193
C05047=1187.048,-75.338,-41.025,179.352,5.658,149.193
C05048=1187.054,-75.608,-41.013,179.350,5.658,149.194
C05049=1187.059,-75.880,-41.002,179.347,5.657,149.195
C05050=1187.065,-76.151,-40.990,179.345,5.658,149.196
C05051=1187.071,-76.400,-40.980,179.342,5.657,149.196
C05052=1187.076,-76.650,-40.969,179.340,5.657,149.197
C05053=1187.081,-76.899,-40.959,179.338,5.657,149.197
C05054=1187.086,-77.149,-40.948,179.335,5.657,149.198
C05055=1187.092,-77.399,-40.938,179.333,5.656,149.199
C05056=1187.096,-77.649,-40.926,179.331,5.656,149.199
C05057=1187.102,-77.898,-40.916,179.328,5.656,149.200
C05058=1187.107,-78.148,-40.906,179.326,5.656,149.201
C05059=1187.112,-78.398,-40.895,179.324,5.655,149.201
C05060=1187.118,-78.648,-40.884,179.321,5.655,149.202
C05061=1187.124,-78.897,-40.873,179.320,5.655,149.202
C05062=1187.129,-79.148,-40.863,179.317,5.655,149.203
C05063=1187.134,-79.397,-40.852,179.315,5.655,149.204
C05064=1187.139,-79.647,-40.841,179.313,5.654,149.204
C05065=1187.144,-79.896,-40.831,179.310,5.654,149.205
C05066=1187.150,-80.146,-40.821,179.308,5.654,149.206
C05067=1187.155,-80.396,-40.810,179.306,5.653,149.206
C05068=1187.160,-80.645,-40.799,179.303,5.653,149.207
C05069=1187.165,-80.895,-40.789,179.301,5.653,149.208
C05070=1187.170,-81.145,-40.779,179.299,5.652,149.208
C05071=1187.175,-81.395,-40.769,179.297,5.653,149.209
C05072=1187.181,-81.644,-40.758,179.294,5.652,149.210
C05073=1187.185,-81.894,-40.747,179.292,5.652,149.210
C05074=1187.191,-82.144,-40.737,179.290,5.652,149.211
C05075=1187.197,-82.393,-40.727,179.287,5.652,149.211
C05076=1187.202,-82.643,-40.716,179.286,5.652,149.212
C05077=1187.207,-82.893,-40.706,179.283,5.651,149.213
C05078=1187.212,-83.143,-40.695,179.280,5.651,149.213
C05079=1187.218,-83.392,-40.684,179.279,5.651,149.214
C05080=1187.223,-83.642,-40.674,179.276,5.650,149.215
C05081=1187.228,-83.892,-40.664,179.274,5.651,149.215
C05082=1187.234,-84.141,-40.653,179.272,5.650,149.216
C05083=1187.239,-84.392,-40.643,179.269,5.650,149.216
C05084=1187.244,-84.641,-40.633,179.267,5.650,149.217
C05085=1187.249,-84.891,-40.623,179.265,5.649,149.218
C05086=1187.254,-85.141,-40.612,179.263,5.650,149.218
C05087=1187.260,-85.390,-40.602,179.261,5.649,149.219
C05088=1187.264,-85.640,-40.591,179.258,5.648,149.220
C05089=1187.270,-85.889,-40.581,179.256,5.649,149.220
C05090=1187.275,-86.140,-40.570,179.254,5.648,149.221
C05091=1187.281,-86.389,-40.560,179.252,5.648,149.221
C05092=1187.286,-86.639,-40.550,179.249,5.648,149.222
C05093=1187.290,-86.889,-40.540,179.247,5.648,149.223
C05094=1187.296,-87.138,-40.530,179.245,5.647,149.223
C05095=1187.302,-87.388,-40.519,179.242,5.647,149.224
C05096=1187.307,-87.638,-40.509,179.240,5.647,149.225
C05097=1187.312,-87.888,-40.499,179.238,5.647,149.225
C05098=1187.318,-88.137,-40.488,179.236,5.647,149.226
C05099=1187.322,-88.387,-40.478,179.234,5.646,149.226
C05100=1187.328,-88.637,-40.468,179.231,5.646,149.227
C05101=1187.333,-88.886,-40.458,179.229,5.646,149.228
C05102=1187.338,-89.136,-40.447,179.227,5.645,149.228
C05103=1187.344,-89.386,-40.437,179.224,5.646,149.229
C05104=1187.350,-89.635,-40.427,179.222,5.645,149.230
C05105=1187.354,-89.885,-40.417,179.220,5.645,149.230
C05106=1187.359,-90.135,-40.407,179.218,5.645,149.231
C05107=1187.365,-90.384,-40.397,179.215,5.644,149.231
C05108=1187.370,-90.635,-40.386,179.213,5.645,149.232
C05109=1187.375,-90.884,-40.376,179.211,5.644,149.233
C05110=1187.381,-91.134,-40.367,179.209,5.644,149.233
C05111=1187.386,-91.384,-40.356,179.206,5.644,149.234
C05112=1187.391,-91.634,-40.346,179.204,5.643,149.235
C05113=1187.397,-91.883,-40.336,179.202,5.643,149.235
C05114=1187.401,-92.133,-40.326,179.199,5.643,149.236
C05115=1187.407,-92.383,-40.316,179.198,5.643,149.236
C05116=1187.412,-92.632,-40.305,179.195,5.643,149.237
C05117=1187.418,-92.882,-40.295,179.194,5.643,149.238
C05118=1187.422,-93.132,-40.285,179.191,5.642,149.238
C05119=1187.428,-93.381,-40.275,179.188,5.642,149.239
C05120=1187.434,-93.632,-40.266,179.187,5.642,149.240
C05121=1187.438,-93.882,-40.256,179.184,5.641,149.240
C05122=1187.444,-94.131,-40.245,179.182,5.642,149.241
C05123=1187.449,-94.381,-40.235,179.180,5.641,149.241
C05124=1187.455,-94.630,-40.225,179.178,5.641,149.242
C05125=1187.459,-94.880,-40.215,179.175,5.641,149.243
C05126=1187.465,-95.130,-40.206,179.173,5.641,149.243
C05127=1187.471,-95.380,-40.195,179.171,5.641,149.244
C05128=1187.475,-95.629,-40.186,179.168,5.640,149.245
C05129=1187.480,-95.879,-40.175,179.166,5.640,149.245
C05130=1187.486,-96.129,-40.165,179.164,5.639,149.246
C05131=1187.491,-96.379,-40.156,179.162,5.640,149.246
C05132=1187.497,-96.628,-40.146,179.159,5.639,149.247
C05133=1187.502,-96.878,-40.135,179.158,5.639,149.248
C05134=1187.507,-97.128,-40.126,179.155,5.639,149.248
C05135=1187.513,-97.378,-40.116,179.154,5.639,149.249
C05136=1187.518,-97.627,-40.106,179.151,5.639,149.250
C05137=1187.522,-97.877,-40.096,179.148,5.638,149.250
C05138=1187.528,-98.127,-40.086,179.147,5.638,149.251
C05139=1187.534,-98.377,-40.076,179.144,5.638,149.251
C05140=1187.539,-98.626,-40.067,179.142,5.638,149.252
C05141=1187.544,-98.876,-40.056,179.140,5.637,149.253
C05142=1187.549,-99.126,-40.046,179.138,5.638,149.253
C05143=1187.555,-99.376,-40.037,179.135,5.637,149.254
C05144=1187.560,-99.625,-40.027,179.133,5.637,149.255
C05145=1187.565,-99.875,-40.017,179.131,5.637,149.255
C05146=1187.571,-100.125,-40.008,179.128,5.636,149.256
C05147=1187.576,-100.375,-39.997,179.126,5.637,149.256
C05148=1187.581,-100.624,-39.987,179.124,5.636,149.257
C05149=1187.587,-100.875,-39.978,179.122,5.636,149.258
C05150=1187.592,-101.124,-39.968,179.120,5.636,149.258
C05151=1187.598,-101.396,-39.958,179.118,5.636,149.259
C05152=1187.603,-101.667,-39.947,179.115,5.636,149.260
C05153=1187.609,-101.938,-39.937,179.112,5.635,149.260
C05154=1187.615,-102.210,-39.925,179.110,5.636,149.261
C05155=1187.620,-102.460,-39.916,179.108,5.635,149.261
C05156=1187.626,-102.709,-39.906,179.106,5.635,149.262
C05157=1187.630,-102.960,-39.897,179.104,5.634,149.263
C05158=1187.636,-103.210,-39.887,179.101,5.634,149.263
C05159=1187.641,-103.459,-39.877,179.099,5.634,149.264
C05160=1187.647,-103.709,-39.867,179.097,5.634,149.265
C05161=1187.652,-103.958,-39.858,179.095,5.634,149.265
C05162=1187.657,-104.208,-39.848,179.093,5.633,149.266
C05163=1187.662,-104.458,-39.838,179.091,5.634,149.267
C05164=1187.668,-104.708,-39.829,179.088,5.633,149.267
C05165=1187.672,-104.958,-39.819,179.086,5.633,149.268
C05166=1187.678,-105.207,-39.809,179.084,5.633,149.268
C05167=1187.683,-105.457,-39.800,179.082,5.633,149.269
C05168=1187.689,-105.707,-39.790,179.079,5.632,149.270
C05169=1187.694,-105.956,-39.781,179.078,5.632,149.270
C05170=1187.700,-106.206,-39.771,179.075,5.632,149.271
C05171=1187.704,-106.457,-39.762,179.073,5.632,149.271
C05172=1187.710,-106.706,-39.751,179.071,5.632,149.272
C05173=1187.715,-106.956,-39.743,179.068,5.631,149.273
C05174=1187.721,-107.206,-39.732,179.066,5.631,149.273
C05175=1187.726,-107.455,-39.723,179.064,5.631,149.274
C05176=1187.731,-107.705,-39.713,179.062,5.631,149.274
C05177=1187.736,-107.955,-39.704,179.060,5.630,149.275
C05178=1187.741,-108.204,-39.695,179.058,5.630,149.276
C05179=1187.747,-108.454,-39.685,179.055,5.630,149.276
C05180=1187.752,-108.703,-39.676,179.053,5.631,149.277
C05181=1187.758,-108.954,-39.666,179.051,5.630,149.278
C05182=1187.763,-109.204,-39.657,179.049,5.630,149.278
C05183=1187.768,-109.454,-39.647,179.047,5.629,149.279
C05184=1187.773,-109.704,-39.638,179.045,5.630,149.279
C05185=1187.778,-109.953,-39.628,179.042,5.629,149.280
C05186=1187.784,-110.203,-39.619,179.040,5.629,149.281
C05187=1187.789,-110.452,-39.609,179.038,5.629,149.281
C05188=1187.795,-110.702,-39.599,179.036,5.629,149.282
C05189=1187.800,-110.952,-39.591,179.033,5.629,149.283
C05190=1187.805,-111.201,-39.581,179.032,5.629,149.283
C05191=1187.811,-111.452,-39.571,179.029,5.628,149.284
C05192=1187.816,-111.701,-39.562,179.028,5.628,149.284
C05193=1187.822,-111.951,-39.552,179.025,5.628,149.285
C05194=1187.827,-112.201,-39.543,179.023,5.628,149.285
C05195=1187.832,-112.450,-39.534,179.021,5.627,149.286
C05196=1187.837,-112.700,-39.524,179.019,5.627,149.287
C05197=1187.843,-112.950,-39.515,179.016,5.627,149.287
C05198=1187.847,-113.199,-39.506,179.015,5.627,149.288
C05199=1187.853,-113.449,-39.496,179.012,5.627,149.289
C05200=1187.859,-113.699,-39.487,179.010,5.627,149.289
C05201=1187.863,-113.949,-39.478,179.008,5.626,149.290
C05202=1187.869,-114.199,-39.468,179.006,5.627,149.290
C05203=1187.874,-114.449,-39.459,179.003,5.626,149.291
C05204=1187.880,-114.698,-39.451,179.001,5.626,149.292
C05205=1187.885,-114.948,-39.440,178.999,5.626,149.292
C05206=1187.890,-115.198,-39.431,178.997,5.626,149.293
C05207=1187.896,-115.448,-39.423,178.995,5.625,149.293
C05208=1187.901,-115.697,-39.412,178.993,5.626,149.294
C05209=1187.906,-115.947,-39.403,178.991,5.625,149.295
C05210=1187.912,-116.197,-39.395,178.989,5.625,149.295
C05211=1187.917,-116.447,-39.385,178.986,5.624,149.296
C05212=1187.922,-116.696,-39.375,178.984,5.625,149.296
C05213=1187.927,-116.946,-39.367,178.982,5.624,149.297
C05214=1187.933,-117.196,-39.358,178.980,5.625,149.298
C05215=1187.939,-117.446,-39.348,178.977,5.624,149.298
C05216=1187.943,-117.695,-39.339,178.976,5.624,149.299
C05217=1187.949,-117.945,-39.330,178.973,5.624,149.300
C05218=1187.954,-118.195,-39.320,178.971,5.624,149.300
C05219=1187.960,-118.445,-39.311,178.969,5.623,149.301
C05220=1187.965,-118.695,-39.302,178.967,5.623,149.301
C05221=1187.970,-118.944,-39.293,178.964,5.623,149.302
C05222=1187.975,-119.194,-39.284,178.963,5.623,149.302
C05223=1187.981,-119.444,-39.274,178.960,5.623,149.303
C05224=1187.986,-119.694,-39.265,178.959,5.623,149.304
C05225=1187.991,-119.944,-39.257,178.956,5.622,149.304
C05226=1187.996,-120.194,-39.248,178.954,5.622,149.305
C05227=1188.002,-120.443,-39.237,178.952,5.622,149.306
C05228=1188.008,-120.693,-39.229,178.950,5.622,149.306
C05229=1188.013,-120.942,-39.220,178.947,5.622,149.307
C05230=1188.018,-121.192,-39.211,178.946,5.622,149.307
C05231=1188.023,-121.442,-39.202,178.943,5.621,149.308
C05232=1188.029,-121.692,-39.193,178.941,5.621,149.308
C05233=1188.034,-121.942,-39.184,178.939,5.621,149.309
C05234=1188.039,-122.192,-39.175,178.937,5.621,149.310
C05235=1188.044,-122.441,-39.165,178.934,5.620,149.310
C05236=1188.049,-122.691,-39.156,178.933,5.620,149.311
C05237=1188.055,-122.941,-39.148,178.930,5.620,149.312
C05238=1188.060,-123.191,-39.138,178.929,5.620,149.312
C05239=1188.066,-123.440,-39.130,178.926,5.620,149.313
C05240=1188.071,-123.690,-39.121,178.924,5.620,149.313
C05241=1188.077,-123.940,-39.112,178.922,5.619,149.314
C05242=1188.082,-124.190,-39.103,178.920,5.619,149.314
C05243=1188.087,-124.440,-39.094,178.917,5.619,149.315
C05244=1188.093,-124.690,-39.084,178.916,5.619,149.316
C05245=1188.098,-124.940,-39.076,178.913,5.619,149.316
C05246=1188.103,-125.190,-39.067,178.912,5.619,149.317
C05247=1188.109,-125.439,-39.058,178.909,5.619,149.318
C05248=1188.114,-125.689,-39.049,178.907,5.618,149.318
C05249=1188.119,-125.938,-39.040,178.905,5.619,149.319
C05250=1188.124,-126.188,-39.031,178.903,5.618,149.319
C05251=1188.130,-126.438,-39.023,178.901,5.618,149.320
C05252=1188.135,-126.688,-39.014,178.899,5.618,149.321
C05253=1188.141,-126.938,-39.004,178.897,5.618,149.321
C05254=1188.146,-127.187,-38.996,178.894,5.617,149.322
C05255=1187.724,-127.198,-39.035,178.890,5.620,149.324
C05256=1187.719,-126.948,-39.044,178.893,5.621,149.323
C05257=1187.713,-126.699,-39.052,178.895,5.621,149.322
C05258=1187.708,-126.449,-39.061,178.897,5.622,149.322
C05259=1187.703,-126.199,-39.070,178.899,5.621,149.321
C05260=1187.698,-125.949,-39.079,178.901,5.622,149.321
C05261=1187.693,-125.699,-39.088,178.903,5.622,149.320
C05262=1187.687,-125.449,-39.097,178.906,5.622,149.319
C05263=1187.682,-125.199,-39.106,178.908,5.622,149.319
C05264=1187.676,-124.950,-39.115,178.910,5.623,149.318
C05265=1187.671,-124.700,-39.124,178.912,5.622,149.318
C05266=1187.666,-124.451,-39.133,178.914,5.623,149.317
C05267=1187.660,-124.201,-39.142,178.916,5.623,149.316
C05268=1187.655,-123.951,-39.150,178.918,5.623,149.316
C05269=1187.650,-123.701,-39.159,178.920,5.623,149.315
C05270=1187.644,-123.452,-39.170,178.922,5.623,149.315
C05271=1187.639,-123.202,-39.178,178.925,5.623,149.314
C05272=1187.634,-122.952,-39.187,178.926,5.623,149.313
C05273=1187.628,-122.703,-39.196,178.929,5.624,149.313
C05274=1187.623,-122.453,-39.205,178.931,5.624,149.312
C05275=1187.618,-122.203,-39.214,178.933,5.624,149.312
C05276=1187.612,-121.953,-39.223,178.935,5.624,149.311
C05277=1187.607,-121.703,-39.232,178.938,5.624,149.310
C05278=1187.602,-121.453,-39.241,178.939,5.624,149.310
C05279=1187.597,-121.203,-39.250,178.942,5.625,149.309
C05280=1187.591,-120.953,-39.259,178.943,5.625,149.309
C05281=1187.586,-120.704,-39.269,178.946,5.625,149.308
C05282=1187.581,-120.454,-39.278,178.948,5.625,149.307
C05283=1187.576,-120.204,-39.287,178.950,5.626,149.307
C05284=1187.570,-119.954,-39.296,178.952,5.625,149.306
C05285=1187.565,-119.705,-39.304,178.955,5.626,149.306
C05286=1187.559,-119.455,-39.314,178.956,5.626,149.305
C05287=1187.554,-119.206,-39.323,178.959,5.626,149.304
C05288=1187.549,-118.956,-39.332,178.961,5.626,149.304
C05289=1187.544,-118.706,-39.341,178.963,5.627,149.303
C05290=1187.538,-118.456,-39.351,178.965,5.627,149.303
C05291=1187.532,-118.206,-39.360,178.968,5.627,149.302
C05292=1187.527,-117.956,-39.368,178.969,5.627,149.301
C05293=1187.522,-117.707,-39.378,178.972,5.627,149.301
C05294=1187.516,-117.457,-39.388,178.973,5.627,149.300
C05295=1187.511,-117.207,-39.396,178.976,5.628,149.300
C05296=1187.506,-116.957,-39.405,178.978,5.628,149.299
C05297=1187.501,-116.708,-39.415,178.980,5.628,149.298
C05298=1187.495,-116.458,-39.424,178.982,5.628,149.298
C05299=1187.490,-116.208,-39.433,178.985,5.628,149.297
C05300=1187.485,-115.958,-39.442,178.986,5.628,149.297
C05301=1187.479,-115.708,-39.452,178.989,5.629,149.296
C05302=1187.474,-115.459,-39.461,178.990,5.629,149.295
C05303=1187.469,-115.209,-39.470,178.993,5.629,149.295
C05304=1187.464,-114.959,-39.479,178.995,5.629,149.294
C05305=1187.458,-114.709,-39.489,178.997,5.630,149.294
C05306=1187.453,-114.459,-39.498,179.000,5.629,149.293
C05307=1187.448,-114.210,-39.507,179.002,5.630,149.292
C05308=1187.442,-113.960,-39.517,179.004,5.630,149.292
C05309=1187.437,-113.710,-39.526,179.006,5.630,149.291
C05310=1187.432,-113.460,-39.535,179.008,5.630,149.290
C05311=1187.427,-113.211,-39.545,179.010,5.631,149.290
C05312=1187.421,-112.961,-39.554,179.012,5.630,149.289
C05313=1187.415,-112.711,-39.564,179.015,5.631,149.289
C05314=1187.411,-112.462,-39.573,179.017,5.631,149.288
C05315=1187.405,-112.212,-39.582,179.019,5.631,149.288
C05316=1187.400,-111.962,-39.592,179.021,5.631,149.287
C05317=1187.395,-111.712,-39.601,179.023,5.632,149.286
C05318=1187.389,-111.463,-39.610,179.025,5.631,149.286
C05319=1187.384,-111.212,-39.620,179.028,5.632,149.285
C05320=1187.379,-110.963,-39.629,179.029,5.632,149.284
C05321=1187.373,-110.713,-39.639,179.032,5.632,149.284
C05322=1187.368,-110.464,-39.648,179.034,5.632,149.283
C05323=1187.363,-110.214,-39.657,179.036,5.633,149.282
C05324=1187.357,-109.964,-39.667,179.038,5.633,149.282
C05325=1187.352,-109.714,-39.676,179.041,5.633,149.281
C05326=1187.346,-109.464,-39.686,179.042,5.633,149.281
C05327=1187.342,-109.214,-39.696,179.045,5.633,149.280
C05328=1187.337,-108.965,-39.705,179.047,5.633,149.280
C05329=1187.331,-108.714,-39.714,179.049,5.634,149.279
C05330=1187.326,-108.465,-39.724,179.052,5.634,149.278
C05331=1187.320,-108.215,-39.733,179.054,5.634,149.278
C05332=1187.315,-107.966,-39.743,179.056,5.634,149.277
C05333=1187.309,-107.716,-39.753,179.058,5.634,149.276
C05334=1187.304,-107.466,-39.762,179.060,5.635,149.276
C05335=1187.299,-107.216,-39.771,179.062,5.635,149.275
C05336=1187.294,-106.967,-39.781,179.065,5.635,149.275
C05337=1187.288,-106.717,-39.790,179.066,5.635,149.274
C05338=1187.283,-106.468,-39.800,179.069,5.636,149.273
C05339=1187.278,-106.217,-39.810,179.071,5.635,149.273
C05340=1187.273,-105.967,-39.820,179.073,5.636,149.272
C05341=1187.268,-105.718,-39.829,179.075,5.636,149.271
C05342=1187.262,-105.468,-39.839,179.078,5.636,149.271
C05343=1187.257,-105.218,-39.848,179.080,5.636,149.270
C05344=1187.251,-104.969,-39.858,179.082,5.637,149.270
C05345=1187.246,-104.719,-39.867,179.084,5.636,149.269
C05346=1187.240,-104.469,-39.877,179.087,5.637,149.268
C05347=1187.236,-104.219,-39.887,179.088,5.637,149.268
C05348=1187.230,-103.969,-39.897,179.091,5.637,149.267
C05349=1187.225,-103.720,-39.906,179.093,5.638,149.267
C05350=1187.219,-103.470,-39.916,179.095,5.638,149.266
C05351=1187.215,-103.221,-39.925,179.097,5.638,149.265
C05352=1187.209,-102.971,-39.936,179.099,5.638,149.265
C05353=1187.204,-102.721,-39.944,179.102,5.638,149.264
C05354=1187.199,-102.471,-39.955,179.104,5.638,149.264
C05355=1187.194,-102.221,-39.964,179.106,5.639,149.263
C05356=1187.188,-101.949,-39.975,179.108,5.638,149.262
C05357=1187.182,-101.678,-39.985,179.111,5.639,149.262
C05358=1187.176,-101.407,-39.996,179.113,5.639,149.261
C05359=1187.170,-101.135,-40.007,179.115,5.639,149.260
C05360=1187.165,-100.885,-40.017,179.118,5.639,149.260
C05361=1187.159,-100.635,-40.026,179.120,5.640,149.259
C05362=1187.155,-100.386,-40.036,179.122,5.640,149.258
C05363=1187.150,-100.136,-40.046,179.125,5.641,149.258
C05364=1187.144,-99.886,-40.056,179.127,5.640,149.257
C05365=1187.139,-99.636,-40.065,179.129,5.641,149.256
C05366=1187.133,-99.387,-40.076,179.131,5.641,149.256
C05367=1187.128,-99.137,-40.085,179.134,5.641,149.255
C05368=1187.123,-98.887,-40.095,179.135,5.641,149.255
C05369=1187.118,-98.637,-40.105,179.138,5.641,149.254
C05370=1187.112,-98.387,-40.114,179.140,5.641,149.253
C05371=1187.107,-98.138,-40.124,179.142,5.642,149.253
C05372=1187.101,-97.888,-40.135,179.145,5.642,149.252
C05373=1187.097,-97.638,-40.145,179.146,5.642,149.252
C05374=1187.091,-97.388,-40.154,179.149,5.643,149.251
C05375=1187.085,-97.139,-40.164,179.151,5.642,149.250
C05376=1187.081,-96.889,-40.174,179.153,5.643,149.250
C05377=1187.076,-96.639,-40.185,179.155,5.643,149.249
C05378=1187.070,-96.389,-40.194,179.158,5.643,149.249
C05379=1187.065,-96.140,-40.204,179.160,5.643,149.248
C05380=1187.059,-95.890,-40.214,179.162,5.643,149.247
C05381=1187.054,-95.641,-40.224,179.165,5.644,149.247
C05382=1187.049,-95.391,-40.234,179.167,5.644,149.246
C05383=1187.043,-95.141,-40.244,179.169,5.645,149.245
C05384=1187.038,-94.891,-40.254,179.171,5.644,149.245
C05385=1187.033,-94.642,-40.263,179.174,5.645,149.244
C05386=1187.028,-94.392,-40.274,179.175,5.645,149.244
C05387=1187.022,-94.142,-40.284,179.178,5.645,149.243
C05388=1187.017,-93.892,-40.293,179.180,5.646,149.242
C05389=1187.012,-93.642,-40.304,179.182,5.645,149.242
C05390=1187.007,-93.392,-40.314,179.185,5.646,149.241
C05391=1187.001,-93.143,-40.324,179.186,5.646,149.240
C05392=1186.996,-92.894,-40.334,179.189,5.646,149.240
C05393=1186.991,-92.643,-40.344,179.191,5.646,149.239
C05394=1186.986,-92.394,-40.354,179.193,5.647,149.239
C05395=1186.980,-92.144,-40.365,179.196,5.647,149.238
C05396=1186.975,-91.894,-40.374,179.198,5.647,149.237
C05397=1186.970,-91.644,-40.384,179.200,5.647,149.237
C05398=1186.964,-91.395,-40.394,179.202,5.647,149.236
C05399=1186.959,-91.145,-40.405,179.205,5.648,149.235
C05400=1186.954,-90.895,-40.415,179.207,5.647,149.235
C05401=1186.949,-90.646,-40.425,179.209,5.648,149.234
C05402=1186.943,-90.396,-40.435,179.212,5.649,149.233
C05403=1186.938,-90.146,-40.446,179.214,5.648,149.233
C05404=1186.933,-89.896,-40.456,179.216,5.649,149.232
C05405=1186.928,-89.647,-40.465,179.218,5.649,149.232
C05406=1186.923,-89.397,-40.476,179.221,5.649,149.231
C05407=1186.917,-89.147,-40.486,179.222,5.649,149.230
C05408=1186.911,-88.898,-40.496,179.225,5.649,149.230
C05409=1186.906,-88.648,-40.507,179.227,5.650,149.229
C05410=1186.902,-88.398,-40.517,179.229,5.650,149.228
C05411=1186.896,-88.149,-40.527,179.232,5.650,149.228
C05412=1186.891,-87.898,-40.537,179.233,5.650,149.227
C05413=1186.885,-87.649,-40.548,179.236,5.651,149.227
C05414=1186.880,-87.399,-40.558,179.239,5.651,149.226
C05415=1186.875,-87.149,-40.568,179.240,5.651,149.225
C05416=1186.870,-86.900,-40.578,179.243,5.651,149.225
C05417=1186.865,-86.650,-40.588,179.245,5.651,149.224
C05418=1186.859,-86.400,-40.599,179.247,5.652,149.223
C05419=1186.854,-86.151,-40.609,179.250,5.652,149.223
C05420=1186.849,-85.900,-40.619,179.252,5.652,149.222
C05421=1186.843,-85.651,-40.630,179.254,5.653,149.222
C05422=1186.838,-85.401,-40.640,179.256,5.652,149.221
C05423=1186.833,-85.151,-40.650,179.258,5.653,149.220
C05424=1186.828,-84.902,-40.660,179.261,5.653,149.220
C05425=1186.823,-84.652,-40.671,179.263,5.653,149.219
C05426=1186.817,-84.402,-40.681,179.265,5.654,149.219
C05427=1186.812,-84.153,-40.692,179.268,5.654,149.218
C05428=1186.807,-83.903,-40.702,179.270,5.654,149.217
C05429=1186.801,-83.653,-40.713,179.272,5.654,149.217
C05430=1186.796,-83.403,-40.723,179.274,5.654,149.216
C05431=1186.791,-83.154,-40.733,179.277,5.655,149.215
C05432=1186.786,-82.903,-40.744,179.279,5.655,149.215
C05433=1186.780,-82.654,-40.754,179.281,5.655,149.214
C05434=1186.775,-82.404,-40.764,179.283,5.655,149.214
C05435=1186.770,-82.155,-40.775,179.286,5.656,149.213
C05436=1186.765,-81.905,-40.785,179.288,5.656,149.212
C05437=1186.760,-81.655,-40.796,179.290,5.656,149.212
C05438=1186.754,-81.406,-40.806,179.293,5.656,149.211
C05439=1186.749,-81.156,-40.816,179.295,5.657,149.210
C05440=1186.744,-80.906,-40.828,179.297,5.657,149.210
C05441=1186.738,-80.657,-40.838,179.300,5.657,149.209
C05442=1186.733,-80.407,-40.848,179.302,5.657,149.208
C05443=1186.728,-80.157,-40.859,179.304,5.658,149.208
C05444=1186.723,-79.907,-40.869,179.306,5.658,149.207
C05445=1186.718,-79.658,-40.880,179.309,5.658,149.206
C05446=1186.713,-79.408,-40.891,179.311,5.658,149.206
C05447=1186.707,-79.158,-40.901,179.313,5.658,149.205
C05448=1186.702,-78.908,-40.911,179.316,5.658,149.204
C05449=1186.697,-78.659,-40.922,179.318,5.659,149.204
C05450=1186.692,-78.409,-40.933,179.320,5.659,149.203
C05451=1186.686,-78.159,-40.943,179.322,5.659,149.203
C05452=1186.681,-77.909,-40.954,179.325,5.660,149.202
C05453=1186.676,-77.660,-40.965,179.327,5.660,149.201
C05454=1186.670,-77.410,-40.975,179.329,5.660,149.201
C05455=1186.665,-77.160,-40.985,179.331,5.660,149.200
C05456=1186.659,-76.911,-40.997,179.334,5.661,149.200
C05457=1186.654,-76.661,-41.007,179.336,5.661,149.199
C05458=1186.649,-76.411,-41.018,179.338,5.661,149.198
C05459=1186.644,-76.162,-41.029,179.341,5.661,149.198
C05460=1186.639,-75.890,-41.040,179.343,5.662,149.197
C05461=1186.632,-75.620,-41.052,179.345,5.661,149.196
C05462=1186.626,-75.348,-41.063,179.348,5.662,149.195
C05463=1186.622,-75.078,-41.075,179.350,5.663,149.195
C05464=1186.616,-74.828,-41.085,179.353,5.663,149.194
C05465=1186.610,-74.578,-41.096,179.355,5.663,149.194
C05466=1186.605,-74.329,-41.107,179.357,5.663,149.193
C05467=1186.600,-74.078,-41.118,179.359,5.663,149.192
C05468=1186.595,-73.829,-41.129,179.362,5.663,149.192
C05469=1186.590,-73.579,-41.139,179.365,5.664,149.191
C05470=1186.584,-73.330,-41.150,179.366,5.664,149.191
C05471=1186.579,-73.080,-41.161,179.369,5.664,149.190
C05472=1186.574,-72.831,-41.171,179.372,5.665,149.189
C05473=1186.568,-72.581,-41.183,179.373,5.665,149.189
C05474=1186.563,-72.331,-41.193,179.376,5.665,149.188
C05475=1186.558,-72.081,-41.204,179.378,5.666,149.187
C05476=1186.553,-71.831,-41.215,179.380,5.666,149.187
C05477=1186.547,-71.582,-41.225,179.383,5.666,149.186
C05478=1186.543,-71.332,-41.237,179.385,5.666,149.185
C05479=1186.536,-71.082,-41.247,179.387,5.666,149.185
C05480=1186.532,-70.833,-41.259,179.390,5.667,149.184
C05481=1186.526,-70.583,-41.269,179.392,5.666,149.183
C05482=1186.521,-70.333,-41.280,179.394,5.667,149.183
C05483=1186.516,-70.083,-41.291,179.397,5.668,149.182
C05484=1186.510,-69.834,-41.302,179.399,5.667,149.182
C05485=1186.505,-69.584,-41.313,179.401,5.668,149.181
C05486=1186.500,-69.335,-41.324,179.404,5.669,149.180
C05487=1186.495,-69.084,-41.334,179.406,5.668,149.180
C05488=1186.490,-68.835,-41.346,179.408,5.669,149.179
C05489=1186.484,-68.585,-41.356,179.410,5.669,149.178
C05490=1186.479,-68.335,-41.368,179.413,5.669,149.178
C05491=1186.474,-68.086,-41.379,179.415,5.670,149.177
C05492=1186.469,-67.836,-41.389,179.417,5.670,149.177
